// TIA Portal project "Blank_project_S71200" (V17)

(* hardware
DEVICE "S7-1200 station_1"  S7-1200 Station
   slot 0: "Rack_0"  S7-1200 Rack  Rack  V1.0
   slot 1: "PLC_1"  CPU 1214C DC/DC/DC  6ES7 214-1AG40-0XB0  V4.5
*)

// ===== PLC "PLC_1"  CPU 1214C DC/DC/DC =====

VAR_GLOBAL   // PLC tag table "Default tag table"
   "System_Byte" AT %MB1 : Byte;
   "FirstScan" AT %M1.0 : Bool;
   "DiagStatusUpdate" AT %M1.1 : Bool;
   "AlwaysTRUE" AT %M1.2 : Bool;
   "AlwaysFALSE" AT %M1.3 : Bool;
   "Clock_Byte" AT %MB0 : Byte;
   "Clock_10Hz" AT %M0.0 : Bool;
   "Clock_5Hz" AT %M0.1 : Bool;
   "Clock_2.5Hz" AT %M0.2 : Bool;
   "Clock_2Hz" AT %M0.3 : Bool;
   "Clock_1.25Hz" AT %M0.4 : Bool;
   "Clock_1Hz" AT %M0.5 : Bool;
   "Clock_0.625Hz" AT %M0.6 : Bool;
   "Clock_0.5Hz" AT %M0.7 : Bool;
END_VAR

VAR_GLOBAL CONSTANT   // PLC tag table "UserDiag_Constants"
   "USERDIAG_IOSYSTEM_1" : Int := 1;   // Index for first IO-System/DP-Mastersystem
   "USERDIAG_DEVICES_PER_IO_SYSTEM_UPPER_LIM" : Int := 5;   // Upper limit of devices/slaves per IO-System/DP-Mastersystem
   "USERDIAG_SLOTS_PER_PLC_UPPER_LIM" : Int := 9;   // max number of local modules
   "USERDIAG_IO_SYSTEMS_UPPER_LIM" : Int := 1;   // Upper limit of IO-Systems/DP-Mastersystems
   "USERDIAG_DEVICES_PER_SCREEN_UPPER_LIM" : Int := 5;   // Upper limit of devices per HMI screen
   "USERDIAG_SLOTS_PER_SCREEN_UPPER_LIM" : Int := 9;   // Upper limit of slots per HMI screen
   "USERDIAG_SLOTS_PER_DEVICE_UPPER_LIM" : Int := 9;   // max number of modules per device
END_VAR

// folder: UserDiag

TYPE "UserDiag_typeSlot"
TITLE = UserDiag_typeSlot
   STRUCT
      hardwareId : Hw_Io := 16#0000;   // Hardware identifier of the module which is inserted in the slot
      state : USInt := 0;   // Status of the device/slave. 1:ok; 2:faulty, 3:lost connection, 4:disabled, 5:problem, 12:was faulty, 13:was lost, 14:was disabled, 15:problem gone
      exists : Bool := FALSE;   // TRUE: Modul is existing
      configured : Bool := FALSE;   // TRUE: Modul is configured
      faulty : Bool := FALSE;   // TRUE: Modul is faulty
      problem : Bool := FALSE;   // TRUE: Modul has a problem
      disabled : Bool := FALSE;   // TRUE: Modul is disabled
      error : Bool := FALSE;   // TRUE: Error in module which is inserted in the slot
   END_STRUCT;
END_TYPE

TYPE "UserDiag_typeDevice"
TITLE = UserDiag_typeDevice
   STRUCT
      hardwareId : Hw_Device := 16#0000;   // Hardware identifier of the device/slave
      number : UInt := 0;   // Profinet device number/Profibus address of the slave
      "name" : String[50];   // Name of the device/slave
      ipAddress : IP_V4;   // IP address of the device
      state : USInt := 0;   // Status of the device/slave. 1:ok; 2:faulty, 3:lost connection, 4:disabled, 5:problem, 12:was faulty, 13:was lost, 14:was disabled, 15:problem gone
      exists : Bool := FALSE;   // TRUE: Device/slave is existing
      configured : Bool := FALSE;   // TRUE: Device/slave is configured
      faulty : Bool := FALSE;   // TRUE: Device/slave is faulty
      problem : Bool := FALSE;   // TRUE: Device/slave has a problem
      disabled : Bool := FALSE;   // TRUE: Device/slave is disabled
      error : Bool := FALSE;   // TRUE: Error in device/slave
      nextDevice : Int;   // device number of next device
      actualConfiguredSlots : Int := 0;   // Number of configured slots in the device/slave
      slots : Array[0.."USERDIAG_SLOTS_PER_DEVICE_UPPER_LIM"] of "UserDiag_typeSlot";   // Slot information of a device/slave
   END_STRUCT;
END_TYPE

TYPE "UserDiag_typeIOSystem"
TITLE = UserDiag_typeIOSystem
   STRUCT
      hardwareId : Hw_IoSystem := 16#0000;   // Hardware identifier of the IO-System/DP-Mastersystem
      number : UInt := 0;   // IO-System/DP-Mastersystem number
      error : Bool := FALSE;   // TRUE: Error in IO-System/DP-Mastersystem
      firstDevice : Int := 0;   // device number (index) of first device in IO System
      lastDevice : Int := 0;   // device number (index) of last device IO System
      actualConfiguredDevices : Int := 0;   // Number of configured devices/slaves in IO-System/DP-Mastersystem
      devices : Array[1.."USERDIAG_DEVICES_PER_IO_SYSTEM_UPPER_LIM"] of "UserDiag_typeDevice";   // Device/Slave information
   END_STRUCT;
END_TYPE

TYPE "UserDiag_typePLC"
TITLE = UserDiag_typePLC
   STRUCT
      hardwareId : Hw_Device := 16#0000;   // Hardware identifier of the PLC
      error : Bool := FALSE;   // TRUE: Error in PLC
      actualConfiguredSlots : Int := 0;   // Number of configured local slots at PLC
      slots : Array[0.."USERDIAG_SLOTS_PER_PLC_UPPER_LIM"] of "UserDiag_typeSlot";   // Information of the PLC slots; index = slotnumber; PLC always at slot 1
   END_STRUCT;
END_TYPE

TYPE "UserDiag_typeActIOSystem"
TITLE = UserDiag_typeActIOSystem
   STRUCT
      actIOSystemNumber : Int := 1;   // Number of actual selected IO-system/DP-Mastersystem
      actIODeviceNumbers : Array[1.."USERDIAG_DEVICES_PER_SCREEN_UPPER_LIM"] of UInt;   // Device numbers/profibus addresses of actual selected IO-System/DP-Mastersystem
      actIODeviceState : Array[1.."USERDIAG_DEVICES_PER_SCREEN_UPPER_LIM"] of USInt;   // State of devices/slaves in actual selected IO-System/DP-Mastersystem
      actDeviceSlotsUsed : Array[0.."USERDIAG_SLOTS_PER_SCREEN_UPPER_LIM"] of Bool;   // Used slots of actual selected device/slave
      actDeviceSlotsState : Array[0.."USERDIAG_SLOTS_PER_SCREEN_UPPER_LIM"] of USInt;   // States of actual selected device/slave
   END_STRUCT;
END_TYPE

TYPE "UserDiag_typeHmiData"
   STRUCT
      actIOSystem : Int := 1;   // Index of actual selected IO-System/DP-Mastersystem
      actDeviceOfScreen : Int := 1;   // Index of selected device/slave on actual Screen
      ioSlotDiagnosticsLoaded : Bool;   // TRUE: Page for slot diagnostics is loaded
      actScreenDevices : Int := 1;   // Actual screennumber for copying device status to HMI
      maxScreensDevices : Int;   // Maximum screennumber for copying device status to HMI
      ackWaitTime : Int;   // Wait time after startup, for auto acknowledge
      ackStates : Bool;   // TRUE: Acknowledge of occurred errors in device/slave
      actIOSystemData : "UserDiag_typeActIOSystem";   // Data of actual IO system
      actDeviceNumber : UInt;   // Actual number/profibus address of device/slave
      actDeviceName : String[50];   // Name of actual selected device/slave
      actIPAddress : IP_V4;   // IP address of the device
      errorAtLowerScreen : Bool;   // Error at lower screen
      errorAtUpperScreen : Bool;   // Error at upper screen
      filterErrorDevices : Bool;   // Filter only fault devices
      ioSystemError : Array[1.."USERDIAG_IO_SYSTEMS_UPPER_LIM"] of Bool;   // Error in IO systems
   END_STRUCT;
END_TYPE

// folder: Standard

DATA_BLOCK "DB_Tags"   // DB1
{ S7_Optimized_Access := 'TRUE' }
VERSION : 0.1
   VAR
      TestNull : Bool;   // Always OFF for commissioning only
      TempBOOL : Bool;   // temporary BOOL
      TempWORD : Word;   // temporary WORD
      TempINT : Int;   // temporary INT
      TempDINT : DInt;   // temporary DINT
      TempREAL : Real;   // temporary REAL
      TempDT : DTL;   // temporary DATE AND TIME
      CPU_LED_Status : Int;   // The status of the CPU LED
      Clock01Sec : Bool;   // Impulse 0.1 second
      ClockSec : Bool;   // Impulse 1 second
      ClockMinute : Bool;   // Impulse 1 minute
      ClockHour : Bool;   // Impulse 1 hour
      ClockBlinkFast : Bool;   // Fast blinking clock
      ClockBlinkSlow : Bool;   // Slow blinking clock
      FirstScanDelayed : Bool;   // First cycle with delay
      AckGlobal_NTrigH : Bool;   // 1/0 edge
      Acknowledge : Bool;   // Acknowledge
      Act_PLC_Date_Time : DTL;   // UTC Zeit / UTC time / Actual system date and time
      Set_PLC_Date_Time : DTL := DTL#2000-01-01-0:0:0;   // UTC Zeit / UTC time / Set system date and time
   END_VAR
BEGIN
END_DATA_BLOCK

// folder: System blocks/Program resources

DATA_BLOCK "tDB_FirstScan"   // DB1000
{ S7_Optimized_Access := 'TRUE' }
AUTHOR : Simatic
FAMILY : IEC
NAME : IEC_TMR
VERSION : 1.0
// stored: InstanceOfName IEC_TIMER
"IEC_TIMER"
BEGIN
END_DATA_BLOCK

DATA_BLOCK "tDB_AckGlobal"   // DB1001
{ S7_Optimized_Access := 'TRUE' }
AUTHOR : Simatic
FAMILY : IEC
NAME : IEC_TMR
VERSION : 1.0
// stored: InstanceOfName IEC_TIMER
"IEC_TIMER"
BEGIN
END_DATA_BLOCK

DATA_BLOCK "tDB_01SecClock"   // DB1002
{ S7_Optimized_Access := 'TRUE' }
AUTHOR : Simatic
FAMILY : IEC
NAME : IEC_TMR
VERSION : 1.0
// stored: InstanceOfName IEC_TIMER
"IEC_TIMER"
BEGIN
END_DATA_BLOCK

DATA_BLOCK "tDB_SecClock"   // DB1003
{ S7_Optimized_Access := 'TRUE' }
AUTHOR : Simatic
FAMILY : IEC
NAME : IEC_TMR
VERSION : 1.0
// stored: InstanceOfName IEC_TIMER
"IEC_TIMER"
BEGIN
END_DATA_BLOCK

DATA_BLOCK "tDB_MinClock"   // DB1004
{ S7_Optimized_Access := 'TRUE' }
AUTHOR : Simatic
FAMILY : IEC
NAME : IEC_TMR
VERSION : 1.0
// stored: InstanceOfName IEC_TIMER
"IEC_TIMER"
BEGIN
END_DATA_BLOCK

DATA_BLOCK "tDB_HourClock"   // DB1005
{ S7_Optimized_Access := 'TRUE' }
AUTHOR : Simatic
FAMILY : IEC
NAME : IEC_TMR
VERSION : 1.0
// stored: InstanceOfName IEC_TIMER
"IEC_TIMER"
BEGIN
END_DATA_BLOCK

// folder: UserDiag

DATA_BLOCK "UserDiag_InstMain"   // DB2000
{ S7_Optimized_Access := 'TRUE' }
VERSION : 0.1
// stored: InstanceOfName UserDiag_Main
"UserDiag_Main"
BEGIN
END_DATA_BLOCK

DATA_BLOCK "UserDiag_DiagnosticsData"   // DB2001
TITLE = Diagosis data DB
{ S7_Optimized_Access := 'TRUE' }
VERSION : 0.1
   VAR
      plcData : "UserDiag_typePLC";   // PLC diagnostics data
      ioSystemData : Array[1.."USERDIAG_IO_SYSTEMS_UPPER_LIM"] of "UserDiag_typeIOSystem";   // IO-System diagnostics data
      startDiag : Bool;   // Startflag for diagnostic
   END_VAR
BEGIN
END_DATA_BLOCK

DATA_BLOCK "UserDiag_HmiData"   // DB2002
{ S7_Optimized_Access := 'TRUE' }
VERSION : 0.1
BEGIN
END_DATA_BLOCK

DATA_BLOCK "UserDiag_InstDiagnosticsStartup"   // DB2005
{ S7_Optimized_Access := 'TRUE' }
VERSION : 0.1
// stored: InstanceOfName UserDiag_Diagnostics
"UserDiag_Diagnostics"
BEGIN
END_DATA_BLOCK

// folder: (top level)

ORGANIZATION_BLOCK "Main"   // OB1, LAD, ProgramCycle
TITLE = "Main Program Sweep (Cycle)"
{ S7_Optimized_Access := 'TRUE' }
VERSION : 0.1
   VAR_INPUT
      Initial_Call : Bool;   // Initial call of this OB
      Remanence : Bool;   // =True, if remanent data are available
   END_VAR
BEGIN
END_ORGANIZATION_BLOCK

// folder: Standard

FUNCTION "0000_General_Functions" : Void   // FC0, FBD
{ S7_Optimized_Access := 'TRUE' }
VERSION : 0.1
   VAR_TEMP
      Busy : Bool;
      Mode : USInt;
      Retval_d_act_dp : Int;
      RetVal : Int;
      temp_firstScan : Bool;   // replace with device specific
      temp_ackGlobal : Bool;   // replace with device specific
   END_VAR
   VAR_TEMP   // added for the SCL form of the ladder/FBD networks
      _w1 : Bool;
      _w2 : Bool;
   END_VAR
BEGIN

REGION Network 1: Allways OFF for commissioning only
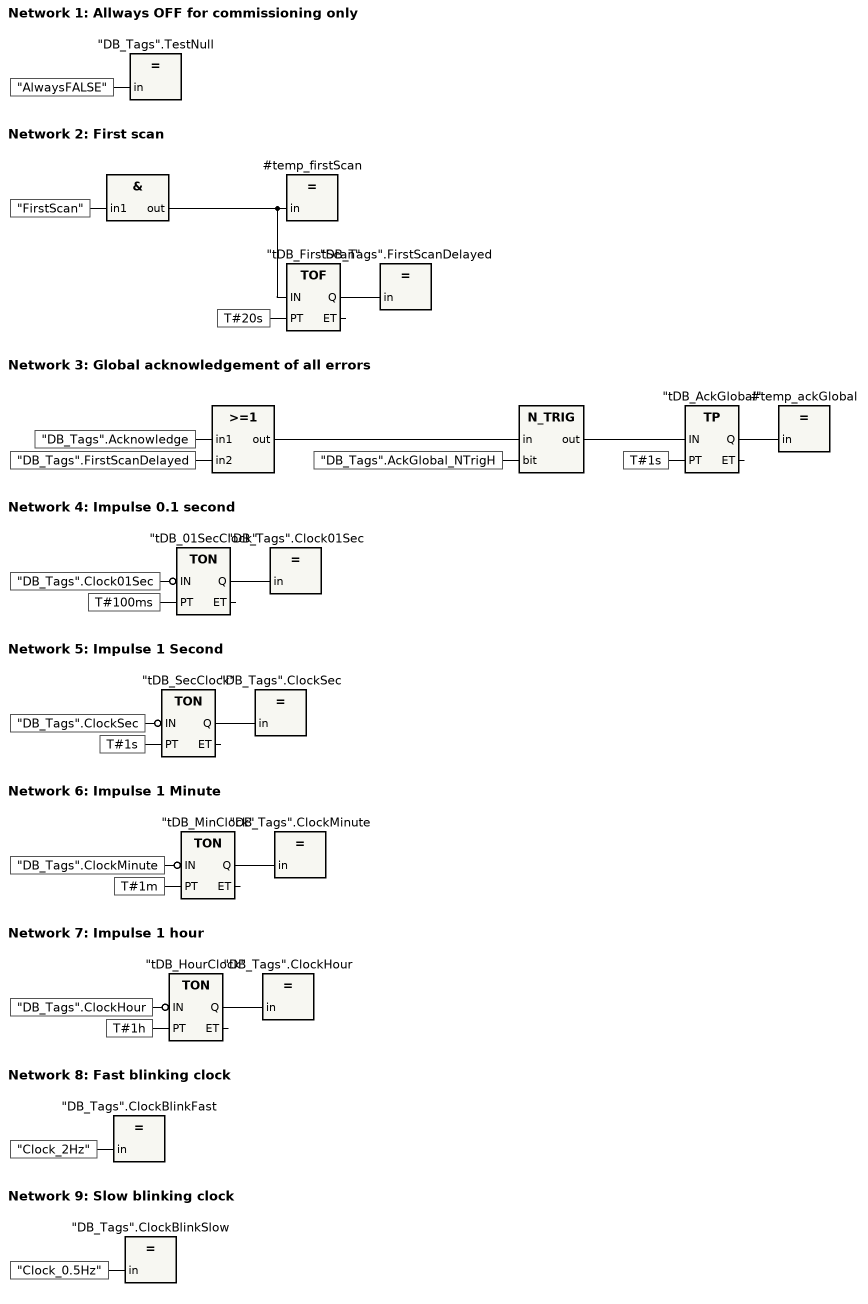
   "DB_Tags".TestNull := "AlwaysFALSE";
END_REGION

REGION Network 2: First scan
   #temp_firstScan := "FirstScan";
   "tDB_FirstScan".TOF(IN := "FirstScan", PT := T#20s);
   "DB_Tags".FirstScanDelayed := "tDB_FirstScan".Q;
END_REGION

REGION Network 3: Global acknowledgement of all errors
   #_w1 := "DB_Tags".Acknowledge OR "DB_Tags".FirstScanDelayed;
   #_w2 := NOT #_w1 AND "DB_Tags".AckGlobal_NTrigH;   // falling edge
   "DB_Tags".AckGlobal_NTrigH := #_w1;
   "tDB_AckGlobal".TP(IN := #_w2, PT := T#1s);
   #temp_ackGlobal := "tDB_AckGlobal".Q;
END_REGION

REGION Network 4: Impulse 0.1 second
   "tDB_01SecClock".TON(IN := NOT "DB_Tags".Clock01Sec, PT := T#100ms);
   "DB_Tags".Clock01Sec := "tDB_01SecClock".Q;
END_REGION

REGION Network 5: Impulse 1 Second
   "tDB_SecClock".TON(IN := NOT "DB_Tags".ClockSec, PT := T#1s);
   "DB_Tags".ClockSec := "tDB_SecClock".Q;
END_REGION

REGION Network 6: Impulse 1 Minute
   "tDB_MinClock".TON(IN := NOT "DB_Tags".ClockMinute, PT := T#1m);
   "DB_Tags".ClockMinute := "tDB_MinClock".Q;
END_REGION

REGION Network 7: Impulse 1 hour
   "tDB_HourClock".TON(IN := NOT "DB_Tags".ClockHour, PT := T#1h);
   "DB_Tags".ClockHour := "tDB_HourClock".Q;
END_REGION

REGION Network 8: Fast blinking clock
   "DB_Tags".ClockBlinkFast := "Clock_2Hz";
END_REGION

REGION Network 9: Slow blinking clock
   "DB_Tags".ClockBlinkSlow := "Clock_0.5Hz";
END_REGION

REGION Network 10: CPU LED status
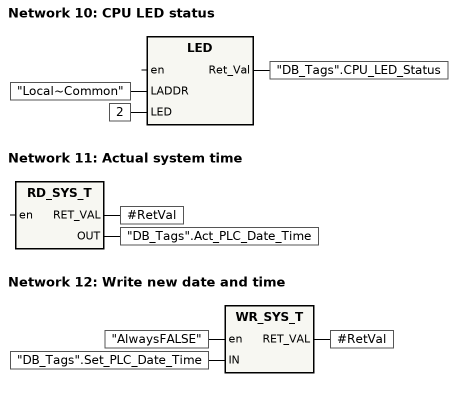
   "DB_Tags".CPU_LED_Status := LED(LADDR := "Local~Common", LED := 2);
END_REGION

REGION Network 11: Actual system time
   #RetVal := RD_SYS_T(OUT => "DB_Tags".Act_PLC_Date_Time);
END_REGION

REGION Network 12: Write new date and time
   IF "AlwaysFALSE" THEN #RetVal := WR_SYS_T(IN := "DB_Tags".Set_PLC_Date_Time); END_IF;
END_REGION
END_FUNCTION

// folder: UserDiag

FUNCTION_BLOCK "UserDiag_Main"   // FB2000, LAD
{ S7_Optimized_Access := 'TRUE' }
VERSION : 0.1
// //============================================================================
// //SIEMENS AG
// //(c)Copyright 2017 All Rights Reserved
// //-----------------------------------------------------------------------------
// //Library: -
// //Tested with: CPU 1214C DC/DC/DC FW4.2
// //Engineering: TIA Portal V15
// //Restrictions: -
// //Requirements: -
// //Functionality: Common FB for diagnostics and HMI
// //-----------------------------------------------------------------------------
// //Change log table:
// //Version  Date              Expert in charge                               Changes applied
// //01.00.00 17.10.2017 Siemens Industry Online Support First released version
// //01.01.00 20.12.2017 Siemens Industry Online Support Call "UserDiag_GetIPAddress"
// //============================================================================
   VAR
      statStartDiag : Bool;   // Static start Diagnostics
      instUserDiagMainDiagnostics : "UserDiag_Diagnostics";   // Instance "UserDiag_MainDiagnostics"
      instUserDiagDiagnosticsHmi : "UserDiag_DiagnosticsHmi";   // Instance "UserDiag_DiagnosticsHmi"
      instUserDiagGetIPAddress : "UserDiag_GetIPAddress";   // Instance "UserDiag_GetIPAddress"
   END_VAR
BEGIN

REGION Network 1: Static start Diagnostics
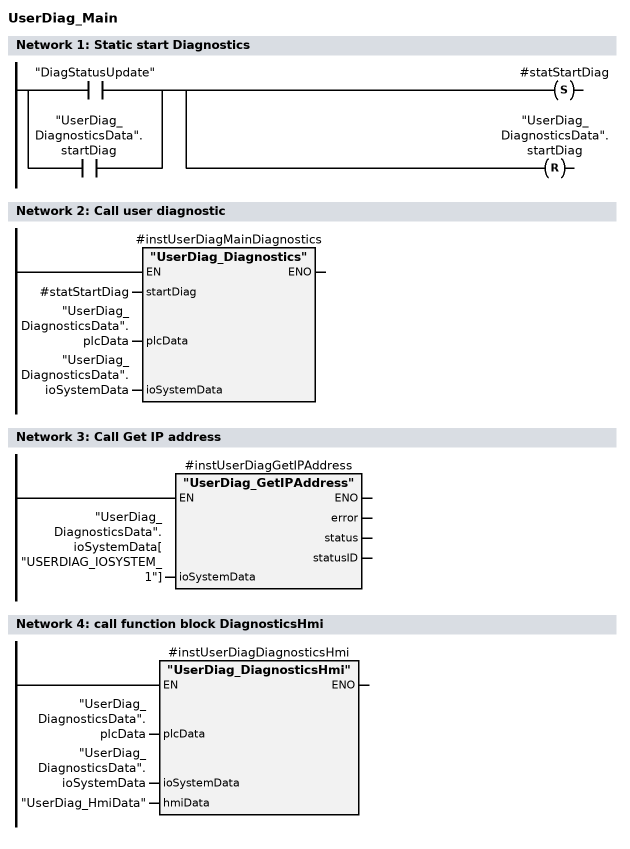
   RUNG wire#powerrail
      Contact( "DiagStatusUpdate" )
      wire#w1
      S_Coil( #statStartDiag )
   END_RUNG
   RUNG wire#powerrail
      Contact( "UserDiag_DiagnosticsData".startDiag )
   END_RUNG wire#w1
   RUNG wire#w1
      R_Coil( "UserDiag_DiagnosticsData".startDiag )
   END_RUNG
   // the same network as SCL:
   IF "DiagStatusUpdate" OR "UserDiag_DiagnosticsData".startDiag THEN
       #statStartDiag := TRUE;
       "UserDiag_DiagnosticsData".startDiag := FALSE;
   END_IF;
END_REGION

REGION Network 2: Call user diagnostic
   RUNG wire#powerrail
      #instUserDiagMainDiagnostics(startDiag := #statStartDiag, plcData := "UserDiag_DiagnosticsData".plcData, ioSystemData := "UserDiag_DiagnosticsData".ioSystemData)
   END_RUNG
   // the same network as SCL:
   #instUserDiagMainDiagnostics(startDiag := #statStartDiag,   // "UserDiag_Diagnostics"
                           plcData := "UserDiag_DiagnosticsData".plcData,
                           ioSystemData := "UserDiag_DiagnosticsData".ioSystemData);
END_REGION

REGION Network 3: Call Get IP address
   RUNG wire#powerrail
      #instUserDiagGetIPAddress(ioSystemData := "UserDiag_DiagnosticsData".ioSystemData["USERDIAG_IOSYSTEM_1"], error =>, status =>, statusID =>)
   END_RUNG
   // the same network as SCL:
   #instUserDiagGetIPAddress(ioSystemData := "UserDiag_DiagnosticsData".ioSystemData["USERDIAG_IOSYSTEM_1"]);   // "UserDiag_GetIPAddress"
END_REGION

REGION Network 4: call function block DiagnosticsHmi
   RUNG wire#powerrail
      #instUserDiagDiagnosticsHmi(plcData := "UserDiag_DiagnosticsData".plcData, ioSystemData := "UserDiag_DiagnosticsData".ioSystemData, hmiData := "UserDiag_HmiData")
   END_RUNG
   // the same network as SCL:
   #instUserDiagDiagnosticsHmi(plcData := "UserDiag_DiagnosticsData".plcData,   // "UserDiag_DiagnosticsHmi"
                           ioSystemData := "UserDiag_DiagnosticsData".ioSystemData,
                           hmiData := "UserDiag_HmiData");
END_REGION
END_FUNCTION_BLOCK

FUNCTION_BLOCK "UserDiag_IOSystemCheck"   // FB2001, SCL
{ S7_Optimized_Access := 'TRUE' }
VERSION : 0.1
   VAR_INPUT
      ioSystemHwId : Hw_IoSystem := 16#0000;   // This ID is representing the IO System (PN or DP), find the ID in the system constants
   END_VAR
   VAR_OUTPUT
      error : Bool := FALSE;   // Rising edge informs that an error occurred during the execution of the FB
      status : Word := 16#0000;   // Current status of FB
      statusID : Word;   // Current status ID of calling instruction
   END_VAR
   VAR_IN_OUT
      ioSystemData : "UserDiag_typeIOSystem";   // IO-System diagnostics data
   END_VAR
   VAR
      statError : Bool := FALSE;   // Static value for output error
      statStatus : Word := 16#0000;   // Static value for output status
      statStatusID : Word;   // Static value for output statusID
      statActualConfiguredDevices : Int := 0;   // Actual number of devices/slaves in the IOSystem/DP-Mastersystem
      statGeoAddr : GEOADDR;   // Slot information
      statGeoLaddr : Hw_Any := 16#0000;   // GEO2LOG hardware identifier
      statConfiguredDevices : Array[0..#DEVICES_STATES_UPPER_LIM] of Bool;   // Temporary storage of the return of "DeviceStates", to combine the states of the devices/slaves with numbers and names
      statExistingDevices : Array[0..#DEVICES_STATES_UPPER_LIM] of Bool;   // Temporary storage of the return of "DeviceStates", to combine the states of the devices/slaves with numbers and names
      statFaultyDevices : Array[0..#DEVICES_STATES_UPPER_LIM] of Bool;   // Temporary storage of the return of "DeviceStates", to combine the states of the devices/slaves with numbers and names
      statDisabledDevices : Array[0..#DEVICES_STATES_UPPER_LIM] of Bool;   // Temporary storage of the return of "DeviceStates", to combine the states of the devices/slaves with numbers and names
      statProblemDevices : Array[0..#DEVICES_STATES_UPPER_LIM] of Bool;   // Temporary storage of the return of "DeviceStates", to combine the states of the devices/slaves with numbers and names
      statDeviceProblemModules : Array[0..#MODULES_STATES_UPPER_LIM] of Bool;   // Storage of the status of all modules in the PN Devices / PB Slaves --> State: Problem
      statDeviceFaultyModules : Array[0..#MODULES_STATES_UPPER_LIM] of Bool;   // Storage of the status of all modules in the PN Devices / PB Slaves --> State: Faulty
      statDeviceExistingModules : Array[0..#MODULES_STATES_UPPER_LIM] of Bool;   // Storage of the status of all modules in the PN Devices / PB Slaves --> State: Existing
      instGetNameDevices : Get_Name;   // Instance of the system function "GetName"
      statInitString : String;   // Used to initialize the temporary string to convert into STRING[50]
      statFirstDevice : UInt;   // Station number of the first device of the list
      statFirstDeviceFlag : Bool := TRUE;   // Help tag for the first device in the linked list
      statLastDevice : UInt;   // Station number of the last device of the list
      statMaxDevices : Int;   // Max devices per IO system
   END_VAR
   VAR_TEMP
      tempIndex : Int;   // Index of configured devices/slaves
      tempDeviceIndex : Int;   // Device/slave index
      tempSlotIndex : Int;   // Slot index
      tempSlotNum : Int;   // Index module number
      tempRetValGeo : Int;   // GEO2LOG error information
      tempRetValDeviceStates : Int;   // DeviceStates error information
      tempRetValModuleStates : Int;   // Return value of the system function "ModuleStates"
      tempStringConvert : String;   // Store the device names temporary here, to convert them into STRING[50]
      tempLastDevice : UInt;   // Temporary storage of the actual index, if it´s the last device --> store it in static
      tempDeviceInit : "UserDiag_typeDevice";   // Initalization of the device/slave diagnostic structure
   END_VAR
   VAR CONSTANT
      STATUS_EXECUTION_FINISHED : Word := 16#0000;   // Execution finished without errors
      ERR_MAX_SLOTS_PER_DEVICE : Word := 16#8400;   // There are more modules configured as defined with the user constant: USERDIAG_SLOTS_PER_DEVICE_UPPER_LIM
      ERR_MAX_DEVICES_PER_IOSYSTEM : Word := 16#8401;   // There are more modules configured as defined with the user constant: USERDIAG_DEVICES_PER_IO_SYTEM_UPPER_LIM
      ID_LOCAL : Word := 1;   // StatusID local
      ID_MODULE_STATES_CONFIGURED : Word := 2;   // StatusID during ModuleStates command (configured mode)
      ID_MODULE_STATES_FAULTY : Word := 3;   // StatusID during ModuleStates command (faulty mode)
      ID_MODULE_STATES_PROBLEM : Word := 4;   // StatusID during ModuleStates command (problem mode)
      ID_MODULE_STATES_EXISTING : Word := 5;   // StatusID during ModuleStates command (existing mode)
      ID_DEVICE_STATES_CONFIGURED : Word := 6;   // StatusID during DeviceStates command (configuration mode)
      ID_DEVICE_STATES_FAULTY : Word := 7;   // StatusID during DeviceStates command (fault mode)
      ID_DEVICE_STATES_PROBLEM : Word := 8;   // StatusID during DeviceStates command (problem mode)
      ID_DEVICE_STATES_EXISTING : Word := 9;   // StatusID during DeviceStates command (existing mode)
      ID_DEVICE_STATES_DISABLED : Word := 10;   // StatusID during DeviceStates command (disable mode)
      ID_GET_NAME : Word := 11;   // StatusID during GET_NAME command
      MODE_CONFIGURED : USInt := 1;   // Used for instruction DeviceStates/ModuleStates, read out all configured devices/slaves
      MODE_FAULTY : USInt := 2;   // Used for instruction DeviceStates/ModuleStates, read out all faulty devices/slaves
      MODE_DISABLED : USInt := 3;   // Used for instruction DeviceStates/ModuleStates, read out all disabled devices/slaves
      MODE_EXIST : USInt := 4;   // Used for instruction DeviceStates/ModuleStates, read out all devices/slaves not reachable
      MODE_PROBLEM : USInt := 5;   // Used for instruction DeviceStates/ModuleStates, read out all devices with several problems
      DEVICE_SLAVE : USInt := 2;   // GEO2LOG structure: HW type = 2
      MODULE_OF_DEVICE : USInt := 4;   // GEO2LOG structure: HW type = 4
      IO_SYSTEM_AREA : USInt := 1;   // GEO2LOG structure: Area = 1
      DP_SYSTEM_AREA : USInt := 2;   // GEO2LOG structure: Area = 2
      STATE_OK : USInt := 1;   // Device/modul state: ok
      STATE_FAULT : USInt := 2;   // Device/modul state: fault
      STATE_LOST_CON : USInt := 3;   // Device/modul state: lost connection
      STATE_DISABLED : USInt := 4;   // Device/modul state: disabled
      STATE_PROBLEM : USInt := 5;   // Device/modul state: problem
      STATE_WAS_FAULT : USInt := 12;   // Device/modul state: was fault
      STATE_WAS_LOST : USInt := 13;   // Device/modul state: connection was lost
      STATE_WAS_DISABLED : USInt := 14;   // Device/modul state: device/slave was disabled
      STATE_PROBLEM_GONE : USInt := 15;   // Device/modul state: had a problem
      MODULES_STATES_UPPER_LIM : Int := 127;   // Upper array limit for output tag of instruction ModuleStates
      DEVICES_STATES_UPPER_LIM : Int := 1023;   // Upper array limit for output tag of instruction DeviceStates
      ERR_HWID_NOT_EXISTENT : Int := 16#8091;   // Hardware identifier of the LADDR parameter does not exist. Check (for example, in the system constants) whether the value for LADDR exists in the project.
      ERR_LADDR_ADDRESS : Int := 16#8092;   // LADDR does not address a PROFINET IO or DP master system.
      POS_FIRST_CHAR : Int := 50;   // Position of first character to be deleted
      NUMBER_CHAR : Int := 204;   // Number of characters to be deleted
      MAX_SLAVES_DP : Int := 127;   // Max number of slaves in a PROFIBUS IO system
      LAST_DEVICE : Int := -1;   // No next device
   END_VAR
BEGIN
   //=============================================================================
   //SIEMENS AG
   //(c)Copyright 2015 All Rights Reserved
   //-----------------------------------------------------------------------------
   //Library: 
   //Tested with: CPU 1214C DC/DC/DC FW4.2
   //Engineering: TIA Portal V15
   //Restrictions: Call in cyclic OB
   //Requirements: -
   //Functionality: Determine hardware identifier and module states from local and
   //               device modules 
   //-----------------------------------------------------------------------------
   //Change log table:
   //Version  Date       Expert in charge                Changes applied
   //01.00.00 27.01.2017 Siemens Industry Online Support First released version
   //01.00.01 20.12.2017 Siemens Industry Online Support GetStationInfo removed
   //01.00.02 27.02.2018 Siemens Industry Online Support Minor corrections
   //=============================================================================

   IF (#ioSystemHwId <> #ioSystemData.hardwareId)
   THEN
     // New IO System detected at input
     #statFirstDeviceFlag := TRUE;
     #statFirstDevice := 1;
     #statLastDevice := 1;

     #statActualConfiguredDevices := 0;
     #tempDeviceIndex := 1;

     #statError := FALSE;
     #statStatus := #STATUS_EXECUTION_FINISHED;
     #statStatusID := 0;
     #ioSystemData.error := FALSE;
     #ioSystemData.hardwareId := #ioSystemHwId;

     // Find out the number of the assigned IO system
     #tempRetValGeo := LOG2GEO(LADDR := #ioSystemHwId,
                               GEOADDR := #statGeoAddr);
     // Set IO system ID
     #ioSystemData.number := #statGeoAddr.IOSYSTEM;

     // Initialize the structure for system function GEO2LOG
     #statGeoAddr.HWTYPE := #DEVICE_SLAVE;   // Hardware type 2: IO device

     // Predefine the type OF IO system. Either Profinet IO or Profibus DP
     IF (#statGeoAddr.AREA = #IO_SYSTEM_AREA)     // Area ID 1: PROFINET IO
     THEN
       #statMaxDevices := "USERDIAG_DEVICES_PER_IO_SYSTEM_UPPER_LIM";
     ELSIF (#statGeoAddr.AREA = #DP_SYSTEM_AREA) // Area ID 2: Profibus DP
     THEN
       IF ("USERDIAG_DEVICES_PER_IO_SYSTEM_UPPER_LIM" > #MAX_SLAVES_DP)
       THEN
         #statMaxDevices := #MAX_SLAVES_DP;
       ELSE
         #statMaxDevices := "USERDIAG_DEVICES_PER_IO_SYSTEM_UPPER_LIM";
       END_IF;
     ELSE
       #statMaxDevices := "USERDIAG_DEVICES_PER_IO_SYSTEM_UPPER_LIM";
     END_IF;

     // Set all other devices to not configured
     FOR #tempIndex := 1 TO "USERDIAG_DEVICES_PER_IO_SYSTEM_UPPER_LIM" DO
       #ioSystemData.devices[#tempIndex] := #tempDeviceInit;
     END_FOR;

     //=============================================================================
     // CONFIGURED DEVICES
     //=============================================================================
     // Find out how much devices are configured in the IO System --> PROFINET IO
     // This number is the maximum number of devices, which will be checked in the
     // following programm
     #tempRetValDeviceStates := DeviceStates(LADDR := #ioSystemHwId,
                                             MODE := #MODE_CONFIGURED,
                                             STATE := #statConfiguredDevices);

     // Check if the block call was successful
     IF (#tempRetValDeviceStates = 0)
     THEN
       // Call ok
       ;
     ELSIF (#tempRetValDeviceStates = #ERR_HWID_NOT_EXISTENT)
       OR (#tempRetValDeviceStates = #ERR_LADDR_ADDRESS)
     THEN
       #ioSystemData.error := TRUE;
       #statStatus := INT_TO_WORD(#tempRetValDeviceStates);
       #statStatusID := #ID_DEVICE_STATES_CONFIGURED;
       #statError := TRUE;
     ELSE
       // Error handling
       #statStatus := INT_TO_WORD(#tempRetValDeviceStates);
       #statStatusID := #ID_DEVICE_STATES_CONFIGURED;
       #statError := TRUE;
     END_IF;

     // Check if further devices are configured
     FOR #tempIndex := 1 TO #DEVICES_STATES_UPPER_LIM DO
       IF (((#statConfiguredDevices[#tempIndex] = TRUE)
         AND (#tempIndex > #statMaxDevices))
         AND (
         ((#statGeoAddr.AREA = #DP_SYSTEM_AREA)
         AND (#tempIndex < #MAX_SLAVES_DP))
         OR (#statGeoAddr.AREA = #IO_SYSTEM_AREA))
         )
       THEN
         // In the IOSystem are more devices configured as defined with the user constant
         #statStatus := #ERR_MAX_DEVICES_PER_IOSYSTEM;
         #statStatusID := #ID_LOCAL;
         #statError := TRUE;
       END_IF;
     END_FOR;

     //=============================================================================
     // Go trough all devices and get the status of the configured
     //=============================================================================
     FOR #tempIndex := 1 TO #statMaxDevices DO
       // The devices are configured --> Read out the logical address and the
       // device name
       IF (#statConfiguredDevices[#tempIndex] = TRUE)
       THEN
         // Store the first configured device for the linked list
         IF (#statFirstDeviceFlag = TRUE)
         THEN
           #statFirstDevice := INT_TO_UINT(#tempIndex);
           #ioSystemData.firstDevice := UINT_TO_INT(#statFirstDevice);
           #statFirstDeviceFlag := FALSE;
           #tempLastDevice := INT_TO_UINT(#tempIndex);
           // It´s not the first bit --> Store the actual index as "next device"
           // in the further one!
         ELSE
           #ioSystemData.devices[#tempLastDevice].nextDevice := #tempIndex;
           #tempLastDevice := INT_TO_UINT(#tempIndex);
         END_IF;
         // Store the index of the last device for the exit condition of the
         // followiing instructions
         #statLastDevice := #tempLastDevice;
         #ioSystemData.lastDevice := UINT_TO_INT(#statLastDevice);

         // Initialize the structure for system function GEO2LOG
         #statGeoAddr.STATION := INT_TO_UINT(#tempIndex); // Station number 
         #statGeoAddr.HWTYPE := #DEVICE_SLAVE;   // Hardware type 2: IO device

         // Read LADDR from devices
         #tempRetValGeo := GEO2LOG(GEOADDR := #statGeoAddr,
                                   LADDR => #statGeoLaddr);
         // Everything is ok!
         IF (#tempRetValGeo = 0)
         THEN
           // Store LADDR from devices in diagnostics data block
           #ioSystemData.devices[#tempIndex].hardwareId := #statGeoLaddr;
           #ioSystemData.devices[#tempIndex].number := INT_TO_UINT(#tempIndex);
           #ioSystemData.devices[#tempIndex].configured := TRUE;

           // Store the device name, if the device is existing
           // Get name is an acyclic instruction. In the startup OB, the
           // instruction has to be repeated until it is done or error
           REPEAT
             // Get device name of each decive in PN System
             #instGetNameDevices(LADDR := #ioSystemHwId,
                                 STATION_NR := #statGeoAddr.STATION,
                                 DATA := #tempStringConvert);

           UNTIL ((#instGetNameDevices.DONE = TRUE)
             OR (#instGetNameDevices.ERROR = TRUE))
           END_REPEAT;

           IF (#instGetNameDevices.ERROR = TRUE)
           THEN
             // Error handling
             #statStatus := #instGetNameDevices.STATUS;
             #statStatusID := #ID_GET_NAME;
             #statError := TRUE;

             // Everything is ok --> Convert the String[254] into String[50]    
           ELSIF (#instGetNameDevices.DONE = TRUE)
           THEN
             // Cut all characters more than 50 to reduce the string length
             #ioSystemData.devices[#tempIndex].name := DELETE(IN := #tempStringConvert,
                                                              L := #NUMBER_CHAR,
                                                              P := #POS_FIRST_CHAR);

             // Initialize the temporary string before next loop
             #tempStringConvert := #statInitString;
           ELSE
             ;
           END_IF;


           //=============================================================================
           // Get the logical address of all modules and store the actual number of
           // modules from each device
           //=============================================================================

           // Initialize the structure for system function GEO2LOG
           #statGeoAddr.HWTYPE := #MODULE_OF_DEVICE;   // Hardware type 4: Module

           FOR #tempSlotNum := 0 TO "USERDIAG_SLOTS_PER_DEVICE_UPPER_LIM" DO
             // Slot number
             #statGeoAddr.SLOT := INT_TO_UINT(#tempSlotNum);
             // read LADDR from modules
             #tempRetValGeo := GEO2LOG(GEOADDR := #statGeoAddr,
                                       LADDR => #statGeoLaddr);
             // check Retval
             IF (#tempRetValGeo = 0)
             THEN
               // Store LADDR from modules in diagnostic data block
               #ioSystemData.devices[#tempIndex].slots[#tempSlotNum].hardwareId := #statGeoLaddr;
               #ioSystemData.devices[#tempIndex].actualConfiguredSlots := #ioSystemData.devices[#tempIndex].actualConfiguredSlots + 1;

               #ioSystemData.devices[#tempIndex].slots[#tempSlotNum].configured := TRUE;

             ELSE
               // If the return value is not 0 --> the device/system/module is
               // not configured --> No error handling
               // set LADDR from modules to 0 in diagnostic data block
               #ioSystemData.devices[#tempIndex].slots[#tempSlotNum].hardwareId := 0;
             END_IF;
           END_FOR;

           // Check if further slots are configured
           #statGeoAddr.SLOT := INT_TO_UINT(#tempSlotNum);

           #tempRetValGeo := GEO2LOG(GEOADDR := #statGeoAddr,
                                     LADDR => #statGeoLaddr);

           IF ((#tempRetValGeo = 0)
             AND (#statGeoLaddr <> 16#0))
           THEN
             // In the PLC are more slots configured as defined with the user constant
             #statStatus := #ERR_MAX_SLOTS_PER_DEVICE;
             #statStatusID := #ID_LOCAL;
             #statError := TRUE;
           END_IF;

           // Increment the actual configured devices, store the state and
           // HW_ID as an numerical value (UINT)
           #statActualConfiguredDevices := #statActualConfiguredDevices + 1;
         ELSE
           ;
         END_IF;

       ELSE
         ; // Device not configured
       END_IF;
     END_FOR;

     #ioSystemData.actualConfiguredDevices := #statActualConfiguredDevices;

     // Mark parameter "Next Device" of the last device in the list
     // --> "Next Device" = negative --> Last device in the list
     #ioSystemData.devices[#statLastDevice].nextDevice := #LAST_DEVICE;

   END_IF; // New IO System detected at input

   #ioSystemData.error := FALSE; // Reset the IO-System error status


   //=============================================================================
   // START DIAGNOSTICS EVALUATION
   //=============================================================================

   //=============================================================================
   // EXISTING DEVICES
   //=============================================================================
   #tempRetValDeviceStates := DeviceStates(LADDR := #ioSystemHwId,
                                           MODE := #MODE_EXIST,
                                           STATE := #statExistingDevices);

   // Check if the block call was successful
   IF (#tempRetValDeviceStates = 0)
   THEN
     // Call ok 
     ;
   ELSIF ((#tempRetValDeviceStates = #ERR_HWID_NOT_EXISTENT)
     OR (#tempRetValDeviceStates = #ERR_LADDR_ADDRESS))
   THEN
     #ioSystemData.error := TRUE;
     #statStatus := INT_TO_WORD(#tempRetValDeviceStates);
     #statStatusID := #ID_DEVICE_STATES_EXISTING;
     #statError := TRUE;
   ELSE
     // Error handling
     #statStatus := INT_TO_WORD(#tempRetValDeviceStates);
     #statStatusID := #ID_DEVICE_STATES_EXISTING;
     #statError := TRUE;
   END_IF;

   //=============================================================================
   // FAULTY DEVICES
   //=============================================================================
   #tempRetValDeviceStates := DeviceStates(LADDR := #ioSystemHwId,
                                           MODE := #MODE_FAULTY,
                                           STATE := #statFaultyDevices);

   // Check if the block call was successful
   IF (#tempRetValDeviceStates = 0)
   THEN
     // Call ok
     ;
   ELSIF ((#tempRetValDeviceStates = #ERR_HWID_NOT_EXISTENT)
     OR (#tempRetValDeviceStates = #ERR_LADDR_ADDRESS))
   THEN
     #ioSystemData.error := TRUE;
     #statStatus := INT_TO_WORD(#tempRetValDeviceStates);
     #statStatusID := #ID_DEVICE_STATES_FAULTY;
     #statError := TRUE;
   ELSE
     // Error handling
     #statStatus := INT_TO_WORD(#tempRetValDeviceStates);
     #statStatusID := #ID_DEVICE_STATES_FAULTY;
     #statError := TRUE;
   END_IF;

   //=============================================================================
   // DISABLED DEVICES
   //=============================================================================
   #tempRetValDeviceStates := DeviceStates(LADDR := #ioSystemHwId,
                                           MODE := #MODE_DISABLED,
                                           STATE := #statDisabledDevices);

   // Check if the block call was successful
   IF (#tempRetValDeviceStates = 0)
   THEN
     // Call ok
     ;
   ELSIF ((#tempRetValDeviceStates = #ERR_HWID_NOT_EXISTENT)
     OR (#tempRetValDeviceStates = #ERR_LADDR_ADDRESS))
   THEN
     #ioSystemData.error := TRUE;
     #statStatus := INT_TO_WORD(#tempRetValDeviceStates);
     #statStatusID := #ID_DEVICE_STATES_DISABLED;
     #statError := TRUE;
   ELSE
     // Error handling
     #statStatus := INT_TO_WORD(#tempRetValDeviceStates);
     #statStatusID := #ID_DEVICE_STATES_DISABLED;
     #statError := TRUE;
   END_IF;

   //=============================================================================
   // PROBLEM DEVICES
   //=============================================================================
   #tempRetValDeviceStates := DeviceStates(LADDR := #ioSystemHwId,
                                           MODE := #MODE_PROBLEM,
                                           STATE := #statProblemDevices);

   // Check if the block call was successful
   IF (#tempRetValDeviceStates = 0)
   THEN
     // Call ok
     ;
   ELSIF ((#tempRetValDeviceStates = #ERR_HWID_NOT_EXISTENT)
     OR (#tempRetValDeviceStates = #ERR_LADDR_ADDRESS))
   THEN
     #ioSystemData.error := TRUE;
     #statStatus := INT_TO_WORD(#tempRetValDeviceStates);
     #statStatusID := #ID_DEVICE_STATES_PROBLEM;
     #statError := TRUE;
   ELSE
     // Error handling
     #statStatus := INT_TO_WORD(#tempRetValDeviceStates);
     #statStatusID := #ID_DEVICE_STATES_PROBLEM;
     #statError := TRUE;
   END_IF;

   //=============================================================================
   // Go through configured devices and check for error
   //=============================================================================
   // Initialize the pointer for the first run 
   #tempDeviceIndex := #ioSystemData.firstDevice;

   WHILE ((#tempDeviceIndex <= "USERDIAG_DEVICES_PER_IO_SYSTEM_UPPER_LIM")
     AND (#tempDeviceIndex > 0))
   DO

     IF (#ioSystemData.devices[#tempDeviceIndex].configured = TRUE)
     THEN

       IF (#statDisabledDevices[#tempDeviceIndex] = TRUE)
       THEN
         //===================
         // Device is disabled
         //===================
         #ioSystemData.devices[#tempDeviceIndex].disabled := TRUE;
         #ioSystemData.devices[#tempDeviceIndex].error := FALSE;
         #ioSystemData.devices[#tempDeviceIndex].faulty := FALSE;
         #ioSystemData.devices[#tempDeviceIndex].problem := FALSE;
         #ioSystemData.devices[#tempDeviceIndex].state := #STATE_DISABLED;

       ELSE
         #ioSystemData.devices[#tempDeviceIndex].disabled := FALSE;

         IF (#statExistingDevices[#tempDeviceIndex] = TRUE)
         THEN
           #ioSystemData.devices[#tempDeviceIndex].exists := TRUE;

           CASE #ioSystemData.devices[#tempDeviceIndex].state OF
             #STATE_WAS_FAULT,
             #STATE_WAS_LOST,
             #STATE_WAS_DISABLED,
             #STATE_PROBLEM_GONE:
               ;
             #STATE_FAULT:
               #ioSystemData.devices[#tempDeviceIndex].state := #STATE_WAS_FAULT;
             #STATE_LOST_CON:
               #ioSystemData.devices[#tempDeviceIndex].state := #STATE_WAS_LOST;
             #STATE_DISABLED:
               #ioSystemData.devices[#tempDeviceIndex].state := #STATE_WAS_DISABLED;
             #STATE_PROBLEM:
               #ioSystemData.devices[#tempDeviceIndex].state := #STATE_PROBLEM_GONE;
             ELSE
               #ioSystemData.devices[#tempDeviceIndex].state := #STATE_OK;
           END_CASE;

         ELSE
           // Device not existent
           #ioSystemData.devices[#tempDeviceIndex].error := TRUE;
           #ioSystemData.error := TRUE;
           #ioSystemData.devices[#tempDeviceIndex].exists := FALSE;
         END_IF; // End: Device exists


         IF (#statFaultyDevices[#tempDeviceIndex] = FALSE)
         THEN
           // Device is not faulty
           #ioSystemData.devices[#tempDeviceIndex].error := FALSE;
           #ioSystemData.devices[#tempDeviceIndex].faulty := FALSE;

           IF (#statProblemDevices[#tempDeviceIndex] = FALSE)
           THEN
             //============================
             // Device has no problem
             //============================
             #ioSystemData.devices[#tempDeviceIndex].error := FALSE;
             #ioSystemData.devices[#tempDeviceIndex].problem := FALSE;
           ELSE
             //============================
             // Device has a problem
             //============================
             #ioSystemData.devices[#tempDeviceIndex].error := TRUE;
             #ioSystemData.error := TRUE;
             #ioSystemData.devices[#tempDeviceIndex].problem := TRUE;
             #ioSystemData.devices[#tempDeviceIndex].state := #STATE_PROBLEM;
           END_IF;

         ELSE
           // Device is faulty, don't matter what happened
           #ioSystemData.devices[#tempDeviceIndex].error := TRUE;
           #ioSystemData.error := TRUE;
           #ioSystemData.devices[#tempDeviceIndex].faulty := TRUE;

           IF (#statProblemDevices[#tempDeviceIndex] = FALSE)
           THEN
             //============================
             // Device has no problem
             //============================
             #ioSystemData.devices[#tempDeviceIndex].problem := FALSE;
           ELSE
             //============================
             // Device has a problem
             //============================
             #ioSystemData.devices[#tempDeviceIndex].problem := TRUE;
           END_IF;

           IF (#statExistingDevices[#tempDeviceIndex] = FALSE)
           THEN
             //==========================
             // Device is lost
             //==========================
             #ioSystemData.devices[#tempDeviceIndex].state := #STATE_LOST_CON;
             #ioSystemData.devices[#tempDeviceIndex].exists := FALSE;
           ELSE
             //==========================
             // Device is faulty
             //==========================
             #ioSystemData.devices[#tempDeviceIndex].state := #STATE_FAULT;
             #ioSystemData.devices[#tempDeviceIndex].exists := TRUE;
           END_IF;
         END_IF; // End: // Device is not faulty

       END_IF;

       //=============================================================================
       // Set module states
       //=============================================================================
       // Check ModuleStates if device has a problem or is faulty
       IF ((#ioSystemData.devices[#tempDeviceIndex].problem = TRUE)
         OR (#ioSystemData.devices[#tempDeviceIndex].faulty = TRUE))
       THEN

         // PROBLEM MODULE
         #tempRetValModuleStates := ModuleStates(LADDR := #ioSystemData.devices[#tempDeviceIndex].hardwareId,
                                                 MODE := #MODE_PROBLEM,
                                                 STATE := #statDeviceProblemModules);

         // Check if the block call was successful
         IF (#tempRetValModuleStates = 0)
         THEN
           // Call ok 
           ;
         ELSIF ((#tempRetValModuleStates = #ERR_HWID_NOT_EXISTENT)
           OR (#tempRetValModuleStates = #ERR_LADDR_ADDRESS))
         THEN
           #ioSystemData.error := TRUE;
           #statStatus := INT_TO_WORD(#tempRetValModuleStates);
           #statStatusID := #ID_MODULE_STATES_PROBLEM;
           #statError := TRUE;
         ELSE
           // Error handling
           #statStatus := INT_TO_WORD(#tempRetValModuleStates);
           #statStatusID := #ID_MODULE_STATES_PROBLEM;
           #statError := TRUE;
         END_IF;

         // FAULTY MODULE
         #tempRetValModuleStates := ModuleStates(LADDR := #ioSystemData.devices[#tempDeviceIndex].hardwareId,
                                                 MODE := #MODE_FAULTY,
                                                 STATE := #statDeviceFaultyModules);

         // Check if the block call was successful
         IF (#tempRetValModuleStates = 0)
         THEN
           // Call ok 
           ;
         ELSIF ((#tempRetValModuleStates = #ERR_HWID_NOT_EXISTENT)
           OR (#tempRetValModuleStates = #ERR_LADDR_ADDRESS))
         THEN
           #ioSystemData.error := TRUE;
           #statStatus := INT_TO_WORD(#tempRetValModuleStates);
           #statStatusID := #ID_MODULE_STATES_FAULTY;
           #statError := TRUE;
         ELSE
           // Error handling
           #statStatus := INT_TO_WORD(#tempRetValModuleStates);
           #statStatusID := #ID_MODULE_STATES_FAULTY;
           #statError := TRUE;
         END_IF;

         // EXISTING MODULE
         #tempRetValModuleStates := ModuleStates(LADDR := #ioSystemData.devices[#tempDeviceIndex].hardwareId,
                                                 MODE := #MODE_EXIST,
                                                 STATE := #statDeviceExistingModules);

         // Check if the block call was successful
         IF (#tempRetValModuleStates = 0)
         THEN
           // Call ok 
           ;
         ELSIF ((#tempRetValModuleStates = #ERR_HWID_NOT_EXISTENT)
           OR (#tempRetValModuleStates = #ERR_LADDR_ADDRESS))
         THEN
           #ioSystemData.error := TRUE;
           #statStatus := INT_TO_WORD(#tempRetValModuleStates);
           #statStatusID := #ID_MODULE_STATES_EXISTING;
           #statError := TRUE;
         ELSE
           // Error handling
           #statStatus := INT_TO_WORD(#tempRetValModuleStates);
           #statStatusID := #ID_MODULE_STATES_EXISTING;
           #statError := TRUE;
         END_IF;
       END_IF;


       FOR #tempSlotIndex := 0 TO "USERDIAG_SLOTS_PER_DEVICE_UPPER_LIM" DO
         IF (#ioSystemData.devices[#tempDeviceIndex].slots[#tempSlotIndex].configured = TRUE)
         THEN
           CASE #ioSystemData.devices[#tempDeviceIndex].slots[#tempSlotIndex].state OF
             #STATE_WAS_FAULT,
             #STATE_WAS_LOST,
             #STATE_WAS_DISABLED,
             #STATE_PROBLEM_GONE:
               ;
             #STATE_FAULT:
               #ioSystemData.devices[#tempDeviceIndex].slots[#tempSlotIndex].state := #STATE_WAS_FAULT;
             #STATE_LOST_CON:
               #ioSystemData.devices[#tempDeviceIndex].slots[#tempSlotIndex].state := #STATE_WAS_LOST;
             #STATE_DISABLED:
               #ioSystemData.devices[#tempDeviceIndex].slots[#tempSlotIndex].state := #STATE_WAS_DISABLED;
             #STATE_PROBLEM:
               #ioSystemData.devices[#tempDeviceIndex].slots[#tempSlotIndex].state := #STATE_PROBLEM_GONE;
             ELSE
               #ioSystemData.devices[#tempDeviceIndex].slots[#tempSlotIndex].state := #STATE_OK;
           END_CASE;
         END_IF;
       END_FOR;

       CASE #ioSystemData.devices[#tempDeviceIndex].state OF

         #STATE_DISABLED:
           FOR #tempSlotIndex := 0 TO "USERDIAG_SLOTS_PER_DEVICE_UPPER_LIM" DO
             IF (#ioSystemData.devices[#tempDeviceIndex].slots[#tempSlotIndex].configured = TRUE)
             THEN
               //NEW: Set all configured modules of device to disabled
               #ioSystemData.devices[#tempDeviceIndex].slots[#tempSlotIndex].disabled := TRUE;
               #ioSystemData.devices[#tempDeviceIndex].slots[#tempSlotIndex].error := FALSE;
               #ioSystemData.devices[#tempDeviceIndex].slots[#tempSlotIndex].faulty := FALSE;
               #ioSystemData.devices[#tempDeviceIndex].slots[#tempSlotIndex].problem := FALSE;
               #ioSystemData.devices[#tempDeviceIndex].slots[#tempSlotIndex].state := #STATE_DISABLED;
             END_IF;
           END_FOR;

         #STATE_LOST_CON:
           // All modules are faulty when connection is lost
           FOR #tempSlotIndex := 0 TO "USERDIAG_SLOTS_PER_DEVICE_UPPER_LIM" DO
             IF (#ioSystemData.devices[#tempDeviceIndex].slots[#tempSlotIndex].configured = TRUE)
             THEN
               #ioSystemData.devices[#tempDeviceIndex].slots[#tempSlotIndex].error := TRUE;
               #ioSystemData.devices[#tempDeviceIndex].slots[#tempSlotIndex].faulty := TRUE;
               #ioSystemData.devices[#tempDeviceIndex].slots[#tempSlotIndex].problem := TRUE;
               #ioSystemData.devices[#tempDeviceIndex].slots[#tempSlotIndex].exists := FALSE;
               #ioSystemData.devices[#tempDeviceIndex].slots[#tempSlotIndex].state := #STATE_LOST_CON;
             END_IF;
           END_FOR;

         #STATE_FAULT,
         #STATE_PROBLEM:
           // The device is reachable, but faulty because of an error in a
           // subordinated system --> check the modules
           // Store the state of the different module in the diag DB
           FOR #tempSlotIndex := 0 TO "USERDIAG_SLOTS_PER_DEVICE_UPPER_LIM" DO
             IF (#ioSystemData.devices[#tempDeviceIndex].slots[#tempSlotIndex].configured = TRUE)
             THEN
               IF (#statDeviceProblemModules[#tempSlotIndex + 1] = TRUE)
               THEN
                 // Problem in module
                 #ioSystemData.devices[#tempDeviceIndex].slots[#tempSlotIndex].faulty := FALSE;
                 #ioSystemData.devices[#tempDeviceIndex].slots[#tempSlotIndex].error := TRUE;
                 #ioSystemData.devices[#tempDeviceIndex].slots[#tempSlotIndex].problem := TRUE;
                 #ioSystemData.devices[#tempDeviceIndex].slots[#tempSlotIndex].state := #STATE_PROBLEM;

                 IF (#statDeviceFaultyModules[#tempSlotIndex + 1] = TRUE)
                 THEN
                   // Fault in module
                   #ioSystemData.devices[#tempDeviceIndex].slots[#tempSlotIndex].faulty := TRUE;
                   #ioSystemData.devices[#tempDeviceIndex].slots[#tempSlotIndex].state := #STATE_FAULT;
                 END_IF;
               ELSE
                 #ioSystemData.devices[#tempDeviceIndex].slots[#tempSlotIndex].error := FALSE;
                 #ioSystemData.devices[#tempDeviceIndex].slots[#tempSlotIndex].problem := FALSE;
                 #ioSystemData.devices[#tempDeviceIndex].slots[#tempSlotIndex].faulty := FALSE;
               END_IF;

               IF (#statDeviceExistingModules[#tempSlotIndex + 1] = TRUE)
               THEN
                 // Module exists
                 #ioSystemData.devices[#tempDeviceIndex].slots[#tempSlotIndex].exists := TRUE;
               ELSE
                 // Module does not exist
                 #ioSystemData.devices[#tempDeviceIndex].slots[#tempSlotIndex].exists := FALSE;
               END_IF;
             END_IF;
           END_FOR;
         ELSE
           // All modules are okay
           FOR #tempSlotIndex := 0 TO "USERDIAG_SLOTS_PER_DEVICE_UPPER_LIM" DO
             IF (#ioSystemData.devices[#tempDeviceIndex].slots[#tempSlotIndex].configured = TRUE)
             THEN
               #ioSystemData.devices[#tempDeviceIndex].slots[#tempSlotIndex].error := FALSE;
               #ioSystemData.devices[#tempDeviceIndex].slots[#tempSlotIndex].problem := FALSE;
               #ioSystemData.devices[#tempDeviceIndex].slots[#tempSlotIndex].faulty := FALSE;
               #ioSystemData.devices[#tempDeviceIndex].slots[#tempSlotIndex].exists := TRUE;
             END_IF;
           END_FOR;
       END_CASE;
     END_IF;

     // Initialize the pointer for the next run
     #tempDeviceIndex := #ioSystemData.devices[#tempDeviceIndex].nextDevice;
   END_WHILE;


   // Write static values to outputs
   #error := #statError;
   #status := #statStatus;
   #statusID := #statStatusID;
END_FUNCTION_BLOCK

FUNCTION_BLOCK "UserDiag_PLCCheck"   // FB2002, SCL
{ S7_Optimized_Access := 'TRUE' }
VERSION : 0.1
   VAR_INPUT
      plcHwId : Hw_Device;   // Hardware ID
   END_VAR
   VAR_OUTPUT
      error : Bool := FALSE;   // Rising edge informs that an error occurred during the execution of the FB
      status : Word := 16#0000;   // Current status of FB
      statusID : Word;   // Current status ID of calling instruction
   END_VAR
   VAR_IN_OUT
      plcData : "UserDiag_typePLC";   // PLC diagnostics data
   END_VAR
   VAR
      statError : Bool := FALSE;   // Static value for output error
      statStatus : Word := 16#0000;   // Static value for output status
      statStatusID : Word;   // Static value for output statusID
      statGeoAddr : GEOADDR;   // Slot information
      statGeoLaddr : Hw_Any := 16#0000;   // GEO2LOG hardware identifier
      statProblemPlcModulStates : Array[0..#MODULES_STATES_UPPER_LIM] of Bool;   // Storage of the status of all modules in the PLC central station --> State: Problem
      statFaultyPlcModulStates : Array[0..#MODULES_STATES_UPPER_LIM] of Bool;   // Storage of the status of all modules in the PLC central station --> State: Faulty
      statExistingPlcModulStates : Array[0..#MODULES_STATES_UPPER_LIM] of Bool;   // Storage of the status of all modules in the PLC central station --> State: Exists
      statActualCentralModules : USInt := 0;   // Actual number of modules in the central station (PLC)
   END_VAR
   VAR_TEMP
      tempSlotNum : Int;   // Index slot number
      tempRetValGeo : Int;   // GEO2LOG error information
      tempRetValModuleStates : Int;   // Return value system function ModuleStates
   END_VAR
   VAR CONSTANT
      STATUS_EXECUTION_FINISHED : Word := 16#0000;   // Execution finished without errors
      ERR_MAX_SLOTS_PER_PLC : Word := 16#8400;   // There are more modules configured as defined with the user constant: USERDIAG_SLOTS_PER_PLC_UPPER_LIM
      ID_LOCAL : Word := 1;   // StatusID local
      ID_MODULE_STATES_CONFIGURED : Word := 2;   // StatusID during ModuleStates command (configured mode)
      ID_MODULE_STATES_FAULTY : Word := 3;   // StatusID during ModuleStates command (faulty mode)
      ID_MODULE_STATES_PROBLEM : Word := 4;   // StatusID during ModuleStates command (problem mode)
      ID_MODULE_STATES_EXISTING : Word := 5;   // StatusID during ModuleStates command (existing mode)
      ID_LED : Word := 12;   // StatusID occurred during LED command
      MODE_FAULTY : USInt := 2;   // Used for instruction DeviceStates, read out all faulty devices
      MODE_EXIST : USInt := 4;   // Used for instruction DeviceStates, read out all devices not reachable
      MODE_PROBLEM : USInt := 5;   // Used for instruction DeviceStates, read out all devices with several problems
      STATE_OK : USInt := 1;   // Module state: ok
      STATE_FAULT : USInt := 2;   // Modulestate: fault
      STATE_PROBLEM : USInt := 5;   // Module state: problem
      STATE_WAS_FAULT : USInt := 12;   // Module state: was fault
      STATE_PROBLEM_GONE : USInt := 15;   // Module state: had a problem
      MODULE_OF_PLC : USInt := 4;   // GEO2LOG structure: HW type = 4
      CPU : USInt := 0;   // GEO2LOG structure: Area = 0
      CENTRAL_SYSTEM : USInt := 0;   // GEO2LOG structure: IO System = 0
      CENTRAL_STATION : USInt := 0;   // GEO2LOG structure: Station = 0
      NO_LED : Int := 0;   // LED does not exist
      LED_OFF : Int := 1;   // LED is permanently switched off
      LED_NO_INFO : Int := 9;   // LED exists, but status information not available
      MODULES_STATES_UPPER_LIM : Int := 127;   // Upper array limit for output tag of instruction ModuleStates
      ERROR_LED : UInt := 2;   // Identification number of the LED
   END_VAR
BEGIN
   //=============================================================================
   //SIEMENS AG
   //(c)Copyright 2017 All Rights Reserved
   //-----------------------------------------------------------------------------
   //Library: 
   //Tested with: CPU 1214C DC/DC/DC FW4.2
   //Engineering: TIA Portal V15
   //Restrictions: Call in cyclic OB
   //Requirements: -
   //Functionality: Determine plc state and local module states
   //-----------------------------------------------------------------------------
   //Change log table:
   //Version  Date       Expert in charge                Changes applied
   //01.00.00 27.01.2017 Siemens Industry Online Support First released version
   //01.00.01 20.12.2017 Siemens Industry Online Support actualConfiguredSlots >= 1
   //01.00.02 27.02.2018 Siemens Industry Online Support Minor corrections
   //=============================================================================

   IF (#plcData.hardwareId = 0)
   THEN
     #statGeoAddr.HWTYPE := #MODULE_OF_PLC;      // Hardware type 4: module
     #statGeoAddr.AREA := #CPU;                  // Area ID 0: CPU
     #statGeoAddr.IOSYSTEM := #CENTRAL_SYSTEM;   // PROFINET IO system (0 = central unit in the rack)
     #statGeoAddr.STATION := #CENTRAL_STATION;   // Number of the rack if area identifier AREA = 0 (central module)

     #statStatus := #STATUS_EXECUTION_FINISHED;
     #statStatusID := 0;
     #statError := FALSE;
     #statActualCentralModules := 0;

     FOR #tempSlotNum := 0 TO "USERDIAG_SLOTS_PER_PLC_UPPER_LIM" DO
       // Slot number
       #statGeoAddr.SLOT := INT_TO_UINT(#tempSlotNum);
       // read LADDR from local modules
       #tempRetValGeo := GEO2LOG(GEOADDR := #statGeoAddr,
                                 LADDR => #statGeoLaddr);
       // Check Retval
       IF ((#tempRetValGeo = 0)
         AND (#statGeoLaddr <> 16#0))
       THEN
         // Store LADDR from local modules in diagnostic data block
         IF (#tempSlotNum = 1)
         THEN
           #plcData.hardwareId := #statGeoLaddr;
         END_IF;
         #plcData.slots[#tempSlotNum].hardwareId := #statGeoLaddr;
         #statActualCentralModules := #statActualCentralModules + 1;
         #plcData.slots[#tempSlotNum].configured := TRUE;
       ELSE
         // If the return value ist not = 0 --> the device/system/module is not
         // configured --> No error handling
         // set LADDR from local modules to 0 in diagnostic data block
         #plcData.slots[#tempSlotNum].hardwareId := 0;
         #plcData.slots[#tempSlotNum].configured := FALSE;
       END_IF;
       // Store the actual configured devices in the diagnostics DB
       #plcData.actualConfiguredSlots := #statActualCentralModules;
     END_FOR;

     // Check if further slots are configured
     #statGeoAddr.SLOT := INT_TO_UINT(#tempSlotNum);

     #tempRetValGeo := GEO2LOG(GEOADDR := #statGeoAddr,
                               LADDR => #statGeoLaddr);

     IF ((#tempRetValGeo = 0)
       AND (#statGeoLaddr <> 16#0))
     THEN
       // In the PLC are more slots configured as defined with the user constant
       #statStatus := #ERR_MAX_SLOTS_PER_PLC;
       #statStatusID := #ID_LOCAL;
       #statError := TRUE;
     END_IF;

   END_IF;

   // Reset PLC error state
   #plcData.error := FALSE;

   //=============================================================================
   // Check modul states from LOCAL MODULES
   //=============================================================================
   // Check if central module are available - at least one module is always
   // configured, the PLC itself
   IF (#plcData.actualConfiguredSlots >= 1)
   THEN

     // Check the status of the local modules
     #tempRetValModuleStates := ModuleStates(LADDR := #plcHwId,
                                             MODE := #MODE_PROBLEM,
                                             STATE := #statProblemPlcModulStates);

     // Check if the block call was successful
     IF (#tempRetValModuleStates <> 0)
     THEN
       // Error handling
       #statStatus := INT_TO_WORD(#tempRetValModuleStates);
       #statStatusID := #ID_MODULE_STATES_PROBLEM;
       #statError := TRUE;
     ELSE
       ; // Everything is ok!
     END_IF;

     #tempRetValModuleStates := ModuleStates(LADDR := #plcHwId,
                                             MODE := #MODE_FAULTY,
                                             STATE := #statFaultyPlcModulStates);

     // Check if the block call was successful
     IF (#tempRetValModuleStates <> 0)
     THEN
       // Error handling
       #statStatus := INT_TO_WORD(#tempRetValModuleStates);
       #statStatusID := #ID_MODULE_STATES_FAULTY;
       #statError := TRUE;
     ELSE
       ; // Everything is ok!
     END_IF;

     #tempRetValModuleStates := ModuleStates(LADDR := #plcHwId,
                                             MODE := #MODE_EXIST,
                                             STATE := #statExistingPlcModulStates);

     // Check if the block call was successful
     IF (#tempRetValModuleStates <> 0)
     THEN
       // Error handling
       #statStatus := INT_TO_WORD(#tempRetValModuleStates);
       #statStatusID := #ID_MODULE_STATES_EXISTING;
       #statError := TRUE;
     ELSE
       ; // Everything is ok!
     END_IF;

   ELSE
     ; // There are no central moduls configured
   END_IF;

   //=============================================================================
   // Set module states of LOCAL MODULES
   //=============================================================================
   #tempSlotNum := 0;
   WHILE (#tempSlotNum <= #plcData.actualConfiguredSlots)
   DO
     IF (#plcData.slots[#tempSlotNum].configured)
     THEN
       IF (#statExistingPlcModulStates[#tempSlotNum + 1] = TRUE)
       THEN
         #plcData.slots[#tempSlotNum].exists := TRUE;
         CASE #plcData.slots[#tempSlotNum].state OF
           #STATE_WAS_FAULT,
           #STATE_PROBLEM_GONE:
             ;
           #STATE_FAULT:
             #plcData.slots[#tempSlotNum].state := #STATE_WAS_FAULT;
           #STATE_PROBLEM:
             #plcData.slots[#tempSlotNum].state := #STATE_PROBLEM_GONE;
           ELSE
             #plcData.slots[#tempSlotNum].state := #STATE_OK;
         END_CASE;
       ELSE
         #plcData.slots[#tempSlotNum].error := TRUE;
         #plcData.error := TRUE;
         #plcData.slots[#tempSlotNum].exists := FALSE;
       END_IF;

       IF (#statFaultyPlcModulStates[#tempSlotNum + 1] = TRUE)
       THEN
         // Modul is faulty
         #plcData.slots[#tempSlotNum].faulty := TRUE;
         #plcData.slots[#tempSlotNum].problem := TRUE;
         #plcData.slots[#tempSlotNum].error := TRUE;
         #plcData.slots[#tempSlotNum].state := #STATE_FAULT;
       ELSIF (#statProblemPlcModulStates[#tempSlotNum + 1] = TRUE)
       THEN
         // Modul has a problem
         #plcData.slots[#tempSlotNum].faulty := FALSE;
         #plcData.slots[#tempSlotNum].problem := TRUE;
         #plcData.slots[#tempSlotNum].error := TRUE;
         #plcData.slots[#tempSlotNum].state := #STATE_PROBLEM;
       ELSE
         // Modul is OK
         #plcData.slots[#tempSlotNum].error := FALSE;
         #plcData.slots[#tempSlotNum].problem := FALSE;
         #plcData.slots[#tempSlotNum].faulty := FALSE;
       END_IF;

       // Error in PLC - Slot = 1, but index must be increased by 1, because of bit 0 = group display
       // --> used index = 2
       IF (#statProblemPlcModulStates[2] = TRUE)
         OR (#statFaultyPlcModulStates[2] = TRUE)
       THEN
         #plcData.error := TRUE;
       END_IF;
     END_IF;

     #tempSlotNum := #tempSlotNum + 1;
   END_WHILE;

   // Write static values to outputs
   #error := #statError;
   #status := #statStatus;
   #statusID := #statStatusID;

   //----------------------------------------------------------------------------------------------
END_FUNCTION_BLOCK

FUNCTION_BLOCK "UserDiag_Diagnostics"   // FB2003, LAD
{ S7_Optimized_Access := 'TRUE' }
VERSION : 0.1
// //============================================================================
// //SIEMENS AG
// //(c)Copyright 2017 All Rights Reserved
// //-----------------------------------------------------------------------------
// //Library: -
// //Tested with: CPU 1214C DC/DC/DC FW4.2
// //Engineering: TIA Portal V15
// //Restrictions: -
// //Requirements: -
// //Functionality: Main FB for diagnostics
// //-----------------------------------------------------------------------------
// //Change log table:
// //Version  Date              Expert in charge                               Changes applied
// //01.00.00 25.04.2017 Siemens Industry Online Support First released version
// //01.01.00 01.12.2017 Siemens Industry Online Support Renamed in "UserDiag_Diagnostics"
// //                                                                                                    Check Flag "startDiag"
// //============================================================================
   VAR_IN_OUT
      startDiag : Bool;   // Startflag for diagnostic
      plcData : "UserDiag_typePLC";   // PLC diagnostics data
      ioSystemData : Array[1.."USERDIAG_IO_SYSTEMS_UPPER_LIM"] of "UserDiag_typeIOSystem";   // IO-System diagnostics data
   END_VAR
   VAR
      instPLCCheck : "UserDiag_PLCCheck";   // Instance of "UserDiag_PLCCheck"
      instIOSystemCheck1 : "UserDiag_IOSystemCheck";   // Instance of "UserDiag_IOSystemCheck"
      instIOSystemCheck2 : "UserDiag_IOSystemCheck";   // Instance of "UserDiag_IOSystemCheck"
   END_VAR
BEGIN

REGION Network 1: Check Startflag for diagnostic
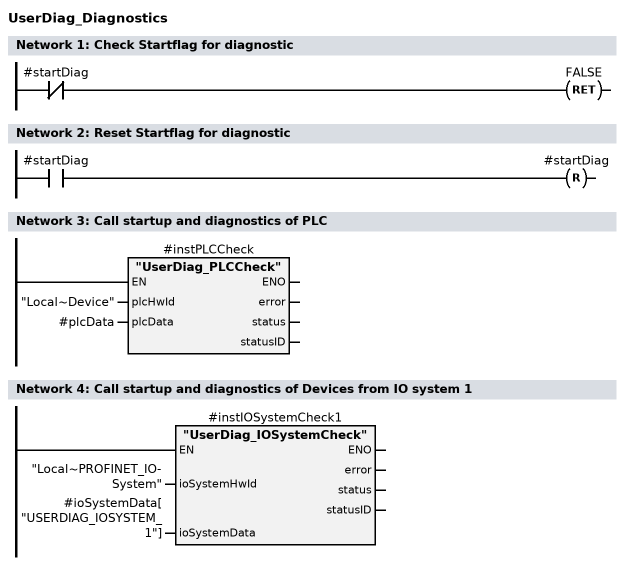
   IF NOT #startDiag THEN
       ENO := FALSE;
       RETURN;
   END_IF;
END_REGION

REGION Network 2: Reset Startflag for diagnostic
   RUNG wire#powerrail
      Contact( #startDiag )
      R_Coil( #startDiag )
   END_RUNG
   // the same network as SCL:
   IF #startDiag THEN #startDiag := FALSE; END_IF;
END_REGION

REGION Network 3: Call startup and diagnostics of PLC
   RUNG wire#powerrail
      #instPLCCheck(plcHwId := "Local~Device", plcData := #plcData, error =>, status =>, statusID =>)
   END_RUNG
   // the same network as SCL:
   #instPLCCheck(plcHwId := "Local~Device", plcData := #plcData);   // "UserDiag_PLCCheck"
END_REGION

REGION Network 4: Call startup and diagnostics of Devices from IO system 1
   RUNG wire#powerrail
      #instIOSystemCheck1(ioSystemHwId := "Local~PROFINET_IO-System", ioSystemData := #ioSystemData["USERDIAG_IOSYSTEM_1"], error =>, status =>, statusID =>)
   END_RUNG
   // the same network as SCL:
   #instIOSystemCheck1(ioSystemHwId := "Local~PROFINET_IO-System",   // "UserDiag_IOSystemCheck"
                       ioSystemData := #ioSystemData["USERDIAG_IOSYSTEM_1"]);
END_REGION
END_FUNCTION_BLOCK

FUNCTION_BLOCK "UserDiag_GetIPAddress"   // FB2005, SCL
{ S7_Optimized_Access := 'TRUE' }
VERSION : 0.1
   VAR_OUTPUT
      error : Bool := FALSE;   // Rising edge informs that an error occurred during the execution of the FB
      status : Word := 16#0000;   // Current status of FB
      statusID : Word;   // Current status ID of calling instruction
   END_VAR
   VAR_IN_OUT
      ioSystemData : "UserDiag_typeIOSystem";   // IO-System diagnostics data
   END_VAR
   VAR
      statError : Bool := FALSE;   // Static value for output error
      statStatus : Word := 16#0000;   // Static value for output status
      statStatusID : Word;   // Static value for output statusID
      instGetStationInfo : GetStationInfo;   // Instance of GetStationInfo
      statFirstDeviceFlag : Bool := TRUE;   // Help tag for the first device in the linked list
      statDeviceIndex : Int;   // Device/slave index
   END_VAR
   VAR_TEMP
      tempIP : IF_CONF_v4;   // Temporary IP address
   END_VAR
   VAR CONSTANT
      STATUS_EXECUTION_FINISHED : Word := 16#0000;   // Execution finished without errors
      ID_GET_STATION_INFO : Word := 12;   // StatusID during GetStationInfo command
      MODE_IPV4 : UInt := 1;   // Address parameter according to IPv4
      LAST_DEVICE : Int := -1;   // No next device
   END_VAR
BEGIN
   //=============================================================================
   //SIEMENS AG
   //(c)Copyright 2015 All Rights Reserved
   //-----------------------------------------------------------------------------
   //Library: 
   //Tested with: CPU 1214C DC/DC/DC FW4.2
   //Engineering: TIA Portal V15
   //Restrictions: Call in cyclic OB
   //Requirements: -
   //Functionality: Get IP address of IO devices
   //-----------------------------------------------------------------------------
   //Change log table:
   //Version  Date       Expert in charge                Changes applied
   //01.00.00 20.12.2017 Siemens Industry Online Support First released version
   //=============================================================================

   //=============================================================================
   // Go through existing devices and get IP address
   //=============================================================================
   // Initialize the pointer for the first run 
   IF (#statFirstDeviceFlag = TRUE)
   THEN
     #statDeviceIndex := #ioSystemData.firstDevice;
     #statFirstDeviceFlag := FALSE;
   END_IF;

   // Check and store the IP address, if the device is existing
   // GetStationInfo is an acyclic instruction. In the FB, the
   // instruction has to be repeated until it is done or error
   IF ((#ioSystemData.number >= 100)
     AND (#ioSystemData.number <= 115)
     AND (#ioSystemData.devices[#statDeviceIndex].exists = TRUE)
     AND (#ioSystemData.devices[#statDeviceIndex].ipAddress.ADDR[1] = 0))
   THEN
     // Get IP address of each decive in PN System
     #instGetStationInfo(REQ := TRUE,
                         LADDR := #ioSystemData.devices[#statDeviceIndex].hardwareId,
                         MODE := #MODE_IPV4,
                         DATA := #tempIP);

     IF (#instGetStationInfo.ERROR = TRUE)
     THEN
       // Error handling
       #statStatus := #instGetStationInfo.STATUS;
       #statStatusID := #ID_GET_STATION_INFO;
       #statError := TRUE;

       // Everything is ok --> Copy IP address    
     ELSIF (#instGetStationInfo.DONE = TRUE)
     THEN
       #ioSystemData.devices[#statDeviceIndex].ipAddress := #tempIP.InterfaceAddress;

       // Initialize the pointer for the next run
       #statDeviceIndex := #ioSystemData.devices[#statDeviceIndex].nextDevice;
     ELSE
       ;
     END_IF;
   ELSE
     // Initialize the pointer for the next run
     #statDeviceIndex := #ioSystemData.devices[#statDeviceIndex].nextDevice;
   END_IF;

   // Check last device
   IF (#statDeviceIndex = #LAST_DEVICE)
   THEN
     #statDeviceIndex := #ioSystemData.firstDevice;
   END_IF;

   // Write static values to outputs
   #error := #statError;
   #status := #statStatus;
   #statusID := #statStatusID;
END_FUNCTION_BLOCK

FUNCTION_BLOCK "UserDiag_DiagnosticsHmi"   // FB2006, SCL
{ S7_Optimized_Access := 'TRUE' }
VERSION : 0.1
   VAR_IN_OUT
      plcData : "UserDiag_typePLC";   // PLC diagnostics data
      ioSystemData : Array[1.."USERDIAG_IO_SYSTEMS_UPPER_LIM"] of "UserDiag_typeIOSystem";   // IO-System diagnostics data
      hmiData : "UserDiag_typeHmiData";   // HMI data
   END_VAR
   VAR
      statFirstRun : Bool := TRUE;   // TRUE after startup
      instAckTON : TON_TIME;   // Instance of TON_TIME for auto acknowledge
      instRisFilterErrorDevices : R_TRIG;   // Instance of R_TRIG for filter error devices
      statActIOSystem : Int;   // Actual IO system
      statActScreenDevices : Int;   // Actual screen devices
      statActDeviceOfScreen : Int;   // Actual device of screen
   END_VAR
   VAR_TEMP
      tempIndex : Int;   // Index of configured devices/slaves
      tempDeviceIndex : Int;   // Device/slave index
      tempDeviceCount : Int;   // Device counter
      tempSlotIndex : Int;   // Slot index
      tempIoIndex : Int;   // IO system index
      tempErrorStateLower : Bool;   // Temp error at lower screen
      tempErrorStateUpper : Bool;   // Temp error at upper screen
   END_VAR
   VAR CONSTANT
      STATE_OK : USInt := 1;   // Device/module state: ok
      STATE_FAULT : USInt := 2;   // Device/modul state: fault
      STATE_LOST_CON : USInt := 3;   // Device/modul state: lost connection
      STATE_DISABLED : USInt := 4;   // Device/modul state: disabled
      STATE_PROBLEM : USInt := 5;   // Device/modul state: problem
      STATE_WAS_FAULT : USInt := 12;   // Device/module state: was fault
      STATE_WAS_LOST : USInt := 13;   // Device/module state: connection was lost
      STATE_WAS_DISABLED : USInt := 14;   // Device/module state: device was disabled
      STATE_PROBLEM_GONE : USInt := 15;   // Device/module state: had a problem
   END_VAR
BEGIN
   //=============================================================================
   //SIEMENS AG
   //(c)Copyright 2017 All Rights Reserved
   //-----------------------------------------------------------------------------
   //Library: 
   //Tested with: CPU 1214C DC/DC/DC FW4.2
   //Engineering: TIA Portal V15
   //Restrictions: Call in cyclic OB
   //Requirements: -
   //Functionality: Copy and control diagnostics information for visualization
   //-----------------------------------------------------------------------------
   //Change log table:
   //Version  Date       Expert in charge                Changes applied
   //01.00.00 27.01.2017 Siemens Industry Online Support First released version
   //01.01.00 17.10.2017 Siemens Industry Online Support Single parameters 
   //                                                    replaced by "hmiData"
   //01.02.00 20.12.2017 Siemens Industry Online Support Static tags for consistence 
   //                                                    (Bereichslängenfehler)
   //=============================================================================

   //=============================================================================
   // Auto acknowledge after waiting time
   //=============================================================================
   #instAckTON(IN := #statFirstRun,
               PT := INT_TO_TIME(#hmiData.ackWaitTime * 1000));

   IF (#instAckTON.Q = TRUE)
   THEN
     // Acknowledge IO systems
     FOR #tempIoIndex := 1 TO "USERDIAG_IO_SYSTEMS_UPPER_LIM" DO
       // Initialize the pointer for the first run 
       #tempDeviceIndex := #ioSystemData[#tempIoIndex].firstDevice;

       WHILE ((#tempDeviceIndex <= "USERDIAG_DEVICES_PER_IO_SYSTEM_UPPER_LIM")
         AND (#tempDeviceIndex > 0))
       DO
         IF (#ioSystemData[#tempIoIndex].devices[#tempDeviceIndex].configured = TRUE)
         THEN
           // Acknowledge "was diabled/faulty/prolem/lost state"
           IF ((#ioSystemData[#tempIoIndex].devices[#tempDeviceIndex].state = #STATE_WAS_DISABLED)
             OR (#ioSystemData[#tempIoIndex].devices[#tempDeviceIndex].state = #STATE_WAS_FAULT)
             OR (#ioSystemData[#tempIoIndex].devices[#tempDeviceIndex].state = #STATE_WAS_LOST)
             OR (#ioSystemData[#tempIoIndex].devices[#tempDeviceIndex].state = #STATE_PROBLEM_GONE))
           THEN
             // Device
             #ioSystemData[#tempIoIndex].devices[#tempDeviceIndex].state := #STATE_OK;
             // Modules
             FOR #tempSlotIndex := 0 TO "USERDIAG_SLOTS_PER_DEVICE_UPPER_LIM" DO
               IF (#ioSystemData[#tempIoIndex].devices[#tempDeviceIndex].slots[#tempSlotIndex].configured = TRUE)
               THEN
                 #ioSystemData[#tempIoIndex].devices[#tempDeviceIndex].slots[#tempSlotIndex].state := #STATE_OK;
               END_IF;
             END_FOR;
           END_IF;
         END_IF;
         // Initialize the pointer for the next run
         #tempDeviceIndex := #ioSystemData[#tempIoIndex].devices[#tempDeviceIndex].nextDevice;
       END_WHILE;

       // Acknowledge local modules
       FOR #tempIndex := 0 TO "USERDIAG_SLOTS_PER_PLC_UPPER_LIM" DO
         IF ((#plcData.slots[#tempIndex].state = #STATE_WAS_FAULT)
           OR (#plcData.slots[#tempIndex].state = #STATE_PROBLEM_GONE))
         THEN
           #plcData.slots[#tempIndex].state := #STATE_OK;
         END_IF;
       END_FOR;
     END_FOR;

     #statFirstRun := FALSE;
   END_IF;

   //=============================================================================
   // Check if a IO system is selected
   //=============================================================================
   // Copy to static tags for consistence
   #statActIOSystem := #hmiData.actIOSystem;
   #statActScreenDevices := #hmiData.actScreenDevices;
   #statActDeviceOfScreen := #hmiData.actDeviceOfScreen;

   IF ((#statActIOSystem >= 1)
     AND (#statActIOSystem <= "USERDIAG_IO_SYSTEMS_UPPER_LIM"))
   THEN
     #hmiData.actIOSystemData.actIOSystemNumber := UINT_TO_INT(#ioSystemData[#statActIOSystem].number);

     // Calculate the maximum count of screens to visualize the devices/slaves
     #hmiData.maxScreensDevices := 1;

     IF ((#ioSystemData[#statActIOSystem].actualConfiguredDevices MOD "USERDIAG_DEVICES_PER_SCREEN_UPPER_LIM") = 0)
     THEN
       #hmiData.maxScreensDevices := #ioSystemData[#statActIOSystem].actualConfiguredDevices / "USERDIAG_DEVICES_PER_SCREEN_UPPER_LIM";
     ELSE
       #hmiData.maxScreensDevices := #ioSystemData[#statActIOSystem].actualConfiguredDevices / "USERDIAG_DEVICES_PER_SCREEN_UPPER_LIM" + 1;
     END_IF;

     //=============================================================================
     // Acknowledge
     //=============================================================================
     IF (#hmiData.ackStates = TRUE)
     THEN
       // Initialize the pointer for the first run 
       #tempDeviceIndex := #ioSystemData[#statActIOSystem].firstDevice;

       WHILE ((#tempDeviceIndex <= "USERDIAG_DEVICES_PER_IO_SYSTEM_UPPER_LIM")
         AND (#tempDeviceIndex > 0))
       DO
         IF (#ioSystemData[#statActIOSystem].devices[#tempDeviceIndex].configured = TRUE)
         THEN
           // Acknowledge "was diabled/faulty/prolem/lost state"
           IF ((#ioSystemData[#statActIOSystem].devices[#tempDeviceIndex].state = #STATE_WAS_DISABLED)
             OR (#ioSystemData[#statActIOSystem].devices[#tempDeviceIndex].state = #STATE_WAS_FAULT)
             OR (#ioSystemData[#statActIOSystem].devices[#tempDeviceIndex].state = #STATE_WAS_LOST)
             OR (#ioSystemData[#statActIOSystem].devices[#tempDeviceIndex].state = #STATE_PROBLEM_GONE))
           THEN
             // Device
             #ioSystemData[#statActIOSystem].devices[#tempDeviceIndex].state := #STATE_OK;
             // Modules
             FOR #tempSlotIndex := 0 TO "USERDIAG_SLOTS_PER_DEVICE_UPPER_LIM" DO
               IF (#ioSystemData[#statActIOSystem].devices[#tempDeviceIndex].slots[#tempSlotIndex].configured = TRUE)
               THEN
                 #ioSystemData[#statActIOSystem].devices[#tempDeviceIndex].slots[#tempSlotIndex].state := #STATE_OK;
               END_IF;
             END_FOR;
           END_IF;
         END_IF;
         // Initialize the pointer for the next run
         #tempDeviceIndex := #ioSystemData[#statActIOSystem].devices[#tempDeviceIndex].nextDevice;
       END_WHILE;
     END_IF;

     //=============================================================================
     // Copy number and status to HMI array
     //=============================================================================
     // Initialize the pointer for the first run 
     #tempDeviceIndex := #ioSystemData[#statActIOSystem].firstDevice;
     // Initialize the pointer for devices on screen
     #tempIndex := 1;
     #tempDeviceCount := 0;

     #instRisFilterErrorDevices(CLK := #hmiData.filterErrorDevices);
     IF (#instRisFilterErrorDevices.Q = TRUE)
     THEN
       #statActScreenDevices := 1;
     END_IF;

     WHILE ((#tempDeviceIndex <= "USERDIAG_DEVICES_PER_IO_SYSTEM_UPPER_LIM")
       AND (#tempDeviceIndex > 0)
       AND (#tempIndex <= "USERDIAG_DEVICES_PER_SCREEN_UPPER_LIM"))
     DO
       IF (#hmiData.filterErrorDevices = FALSE)
       THEN
         IF (#ioSystemData[#statActIOSystem].devices[#tempDeviceIndex].configured = TRUE)
         THEN
           #tempDeviceCount := #tempDeviceCount + 1;

           IF ((#tempDeviceCount > ((#statActScreenDevices - 1) * "USERDIAG_DEVICES_PER_SCREEN_UPPER_LIM"))
             AND (#tempDeviceCount <= (#statActScreenDevices * "USERDIAG_DEVICES_PER_SCREEN_UPPER_LIM")))
           THEN
             // Device configured, status can be copied
             #hmiData.actIOSystemData.actIODeviceNumbers[#tempIndex] := #ioSystemData[#statActIOSystem].devices[#tempDeviceIndex].number;
             #hmiData.actIOSystemData.actIODeviceState[#tempIndex] := #ioSystemData[#statActIOSystem].devices[#tempDeviceIndex].state;
             // Increment index of device per screen
             #tempIndex := #tempIndex + 1;

           END_IF;
         END_IF;
         // Initialize the pointer for the next run
         #tempDeviceIndex := #ioSystemData[#statActIOSystem].devices[#tempDeviceIndex].nextDevice;

         //=============================================================================
         // If filter is enabled, copy number and status of faulty devices to HMI array
         //=============================================================================
       ELSIF (#hmiData.filterErrorDevices = TRUE)
       THEN
         IF ((#ioSystemData[#statActIOSystem].devices[#tempDeviceIndex].configured = TRUE)
           AND (#ioSystemData[#statActIOSystem].devices[#tempDeviceIndex].state > 1))
         THEN
           #tempDeviceCount := #tempDeviceCount + 1;

           IF ((#tempDeviceCount > ((#statActScreenDevices - 1) * "USERDIAG_DEVICES_PER_SCREEN_UPPER_LIM"))
             AND (#tempDeviceCount <= (#statActScreenDevices * "USERDIAG_DEVICES_PER_SCREEN_UPPER_LIM")))
           THEN
             // Device configured, status can be copied
             #hmiData.actIOSystemData.actIODeviceNumbers[#tempIndex] := #ioSystemData[#statActIOSystem].devices[#tempDeviceIndex].number;
             #hmiData.actIOSystemData.actIODeviceState[#tempIndex] := #ioSystemData[#statActIOSystem].devices[#tempDeviceIndex].state;
             // Increment index of device per screen
             #tempIndex := #tempIndex + 1;

           END_IF;
         END_IF;
         // Initialize the pointer for the next run
         #tempDeviceIndex := #ioSystemData[#statActIOSystem].devices[#tempDeviceIndex].nextDevice;

       END_IF;
     END_WHILE;

     // clear screen
     FOR #tempIndex := #tempIndex TO "USERDIAG_DEVICES_PER_SCREEN_UPPER_LIM" DO
       // No device configured
       #hmiData.actIOSystemData.actIODeviceNumbers[#tempIndex] := 0;
       #hmiData.actIOSystemData.actIODeviceState[#tempIndex] := 0;
     END_FOR;

     // Popup for device diagnostics
     IF ((#hmiData.ioSlotDiagnosticsLoaded = TRUE)
       AND (#statActDeviceOfScreen >= 1)
       AND (#statActDeviceOfScreen <= "USERDIAG_DEVICES_PER_SCREEN_UPPER_LIM"))
     THEN
       #tempDeviceIndex := UINT_TO_INT(#hmiData.actIOSystemData.actIODeviceNumbers[#statActDeviceOfScreen]);
       #hmiData.actDeviceName := #ioSystemData[#statActIOSystem].devices[#tempDeviceIndex].name;
       #hmiData.actDeviceNumber := #ioSystemData[#statActIOSystem].devices[#tempDeviceIndex].number;
       #hmiData.actIPAddress := #ioSystemData[#statActIOSystem].devices[#tempDeviceIndex].ipAddress;

       FOR #tempIndex := 0 TO "USERDIAG_SLOTS_PER_SCREEN_UPPER_LIM" DO
         IF (#tempIndex <= "USERDIAG_SLOTS_PER_DEVICE_UPPER_LIM")
         THEN
           #hmiData.actIOSystemData.actDeviceSlotsUsed[#tempIndex] := (#ioSystemData[#statActIOSystem].devices[#tempDeviceIndex].slots[#tempIndex].configured);
           #hmiData.actIOSystemData.actDeviceSlotsState[#tempIndex] := #ioSystemData[#statActIOSystem].devices[#tempDeviceIndex].slots[#tempIndex].state;
         ELSE
           #hmiData.actIOSystemData.actDeviceSlotsUsed[#tempIndex] := FALSE;
           #hmiData.actIOSystemData.actDeviceSlotsState[#tempIndex] := 0;
         END_IF;
       END_FOR;
     END_IF;
     //===============================================================================================================
     // Colors the button, which switches the actual Screen of Devices in case of faulty Device is on different Screen
     //===============================================================================================================
     #tempIndex := 1;
     #tempErrorStateLower := FALSE;
     // Check if devices before the shown in actual Screen are faulty
     WHILE (#tempIndex <= (#hmiData.actIOSystemData.actIODeviceNumbers[1] - 1))
     DO
       IF ((#ioSystemData[#statActIOSystem].devices[#tempIndex].state = #STATE_FAULT)
         OR (#ioSystemData[#statActIOSystem].devices[#tempIndex].state = #STATE_LOST_CON)
         OR (#ioSystemData[#statActIOSystem].devices[#tempIndex].state = #STATE_PROBLEM))
       THEN
         #tempErrorStateLower := TRUE;
       END_IF;
       #tempIndex := #tempIndex + 1;
     END_WHILE;

     #hmiData.errorAtLowerScreen := #tempErrorStateLower;

     #tempIndex := UINT_TO_INT(#hmiData.actIOSystemData.actIODeviceNumbers["USERDIAG_DEVICES_PER_SCREEN_UPPER_LIM"] + 1);
     #tempErrorStateUpper := FALSE;
     // Check if devices after the shown in actual Screen are faulty
     IF (#tempIndex > 1)
     THEN
       WHILE ((#tempIndex <= #ioSystemData[#statActIOSystem].lastDevice))
       DO
         IF ((#ioSystemData[#statActIOSystem].devices[#tempIndex].state = #STATE_FAULT)
           OR (#ioSystemData[#statActIOSystem].devices[#tempIndex].state = #STATE_LOST_CON)
           OR (#ioSystemData[#statActIOSystem].devices[#tempIndex].state = #STATE_PROBLEM))
         THEN
           #tempErrorStateUpper := TRUE;
         END_IF;
         #tempIndex := #tempIndex + 1;
       END_WHILE;
     END_IF;

     #hmiData.errorAtUpperScreen := #tempErrorStateUpper;
     //=============================================================================
     // Check if PLC diagnostics is selected
     //=============================================================================
   ELSIF (#statActIOSystem = -1)
   THEN
     //=============================================================================
     // Acknowledge
     //=============================================================================
     IF (#hmiData.ackStates = TRUE)
     THEN
       FOR #tempIndex := 0 TO "USERDIAG_SLOTS_PER_SCREEN_UPPER_LIM" DO
         IF (#tempIndex <= "USERDIAG_SLOTS_PER_PLC_UPPER_LIM")
         THEN
           IF ((#plcData.slots[#tempIndex].state = #STATE_WAS_FAULT)
             OR (#plcData.slots[#tempIndex].state = #STATE_PROBLEM_GONE))
           THEN
             #plcData.slots[#tempIndex].state := #STATE_OK;
           END_IF;
         END_IF;
       END_FOR;
     END_IF;

     //=============================================================================
     // Copy PLC diagnostics to HMI
     //=============================================================================
     FOR #tempIndex := 0 TO "USERDIAG_SLOTS_PER_SCREEN_UPPER_LIM" DO

       IF (#tempIndex <= "USERDIAG_SLOTS_PER_PLC_UPPER_LIM")
       THEN
         #hmiData.actIOSystemData.actDeviceSlotsUsed[#tempIndex] := (#plcData.slots[#tempIndex].configured);
         #hmiData.actIOSystemData.actDeviceSlotsState[#tempIndex] := #plcData.slots[#tempIndex].state;
       ELSE
         #hmiData.actIOSystemData.actDeviceSlotsUsed[#tempIndex] := FALSE;
         #hmiData.actIOSystemData.actDeviceSlotsState[#tempIndex] := 0;
       END_IF;
     END_FOR;

   ELSE
     ; // No copy of IO System necessary
   END_IF;


   // Set Bit in HMI, if an Error occurs in IO System
   FOR #tempIoIndex := 1 TO "USERDIAG_IO_SYSTEMS_UPPER_LIM" DO
     #hmiData.ioSystemError[#tempIoIndex] := #ioSystemData[#tempIoIndex].error;
   END_FOR;
END_FUNCTION_BLOCK

ORGANIZATION_BLOCK "Startup"   // OB100, LAD, Startup
TITLE = "Complete Restart"
{ S7_Optimized_Access := 'TRUE' }
VERSION : 0.1
// //============================================================================
// //SIEMENS AG
// //(c)Copyright 2017 All Rights Reserved
// //-----------------------------------------------------------------------------
// //Library: -
// //Tested with: CPU 1214C DC/DC/DC FW4.2
// //Engineering: TIA Portal V15
// //Restrictions: -
// //Requirements: -
// //Functionality: Startup OB for Diagnostics
// //-----------------------------------------------------------------------------
// //Change log table:
// //Version  Date              Expert in charge                               Changes applied
// //01.00.00 25.04.2017 Siemens Industry Online Support First released version
// //============================================================================
   VAR_INPUT
      LostRetentive : Bool;   // True if retentive data are lost
      LostRTC : Bool;   // True if date and time are lost
   END_VAR
BEGIN

REGION Network 1: Set start user diagnostic
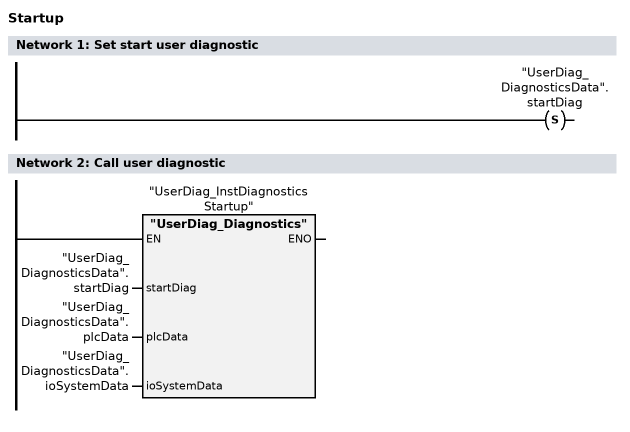
   RUNG wire#powerrail
      S_Coil( "UserDiag_DiagnosticsData".startDiag )
   END_RUNG
   // the same network as SCL:
   "UserDiag_DiagnosticsData".startDiag := TRUE;
END_REGION

REGION Network 2: Call user diagnostic
   RUNG wire#powerrail
      "UserDiag_InstDiagnosticsStartup"(startDiag := "UserDiag_DiagnosticsData".startDiag, plcData := "UserDiag_DiagnosticsData".plcData, ioSystemData := "UserDiag_DiagnosticsData".ioSystemData)
   END_RUNG
   // the same network as SCL:
   "UserDiag_InstDiagnosticsStartup"(startDiag := "UserDiag_DiagnosticsData".startDiag,   // "UserDiag_Diagnostics"
                           plcData := "UserDiag_DiagnosticsData".plcData,
                           ioSystemData := "UserDiag_DiagnosticsData".ioSystemData);
END_REGION
END_ORGANIZATION_BLOCK